C03633=1044.211,253.649,394.364,171.588,39.831,157.569
C03634=1044.205,253.401,394.394,171.585,39.829,157.568
C03635=1044.198,253.153,394.423,171.583,39.827,157.567
C03636=1044.192,252.904,394.453,171.579,39.824,157.567
C03637=1044.185,252.656,394.482,171.576,39.822,157.566
C03638=1044.179,252.408,394.511,171.574,39.820,157.566
C03639=1044.171,252.160,394.540,171.571,39.817,157.565
C03640=1044.165,251.912,394.569,171.568,39.815,157.564
C03641=1044.159,251.664,394.598,171.566,39.812,157.564
C03642=1044.152,251.416,394.627,171.563,39.810,157.563
C03643=1044.146,251.167,394.657,171.561,39.808,157.563
C03644=1044.139,250.919,394.686,171.557,39.806,157.562
C03645=1044.133,250.671,394.715,171.554,39.803,157.561
C03646=1044.126,250.422,394.744,171.552,39.801,157.561
C03647=1044.120,250.174,394.773,171.549,39.798,157.560
C03648=1044.113,249.926,394.802,171.546,39.796,157.560
C03649=1044.107,249.678,394.831,171.544,39.794,157.559
C03650=1044.100,249.430,394.860,171.541,39.791,157.558
C03651=1044.093,249.147,394.894,171.539,39.789,157.558
C03652=1044.085,248.864,394.926,171.535,39.786,157.557
C03653=1044.078,248.581,394.960,171.532,39.784,157.556
C03654=1044.071,248.298,394.992,171.530,39.781,157.556
C03655=1044.064,248.050,395.022,171.527,39.778,157.555
C03656=1044.058,247.802,395.051,171.523,39.776,157.554
C03657=1044.052,247.554,395.080,171.521,39.773,157.554
C03658=1044.046,247.305,395.109,171.518,39.771,157.553
C03659=1044.039,247.057,395.138,171.515,39.769,157.553
C03660=1044.032,246.809,395.166,171.513,39.767,157.552
C03661=1044.025,246.561,395.196,171.510,39.764,157.551
C03662=1044.019,246.313,395.225,171.508,39.762,157.551
C03663=1044.013,246.064,395.254,171.505,39.759,157.550
C03664=1044.007,245.816,395.282,171.502,39.757,157.550
C03665=1044.001,245.568,395.311,171.500,39.755,157.549
C03666=1043.994,245.320,395.339,171.497,39.752,157.548
C03667=1043.987,245.071,395.369,171.495,39.750,157.548
C03668=1043.981,244.823,395.398,171.492,39.747,157.547
C03669=1043.974,244.574,395.426,171.489,39.745,157.547
C03670=1043.968,244.326,395.455,171.487,39.743,157.546
C03671=1043.961,244.078,395.484,171.484,39.741,157.545
C03672=1043.955,243.830,395.511,171.482,39.738,157.545
C03673=1043.949,243.581,395.540,171.479,39.736,157.544
C03674=1043.941,243.333,395.569,171.477,39.734,157.544
C03675=1043.935,243.085,395.598,171.474,39.731,157.543
C03676=1043.929,242.836,395.627,171.471,39.729,157.542
C03677=1043.922,242.588,395.655,171.469,39.726,157.542
C03678=1043.916,242.340,395.683,171.466,39.724,157.541
C03679=1043.909,242.092,395.712,171.464,39.722,157.541
C03680=1043.903,241.844,395.741,171.461,39.720,157.540
C03681=1043.896,241.595,395.769,171.458,39.717,157.539
C03682=1043.890,241.347,395.798,171.456,39.715,157.539
C03683=1043.883,241.099,395.827,171.453,39.713,157.538
C03684=1043.876,240.850,395.855,171.451,39.711,157.538
C03685=1043.869,240.602,395.883,171.448,39.708,157.537
C03686=1043.863,240.353,395.912,171.445,39.706,157.537
C03687=1043.856,240.105,395.940,171.443,39.704,157.536
C03688=1043.850,239.857,395.968,171.440,39.701,157.535
C03689=1043.844,239.608,395.996,171.438,39.699,157.535
C03690=1043.837,239.360,396.024,171.435,39.696,157.534
C03691=1043.830,239.112,396.052,171.432,39.694,157.534
C03692=1043.824,238.864,396.081,171.430,39.692,157.533
C03693=1043.817,238.615,396.109,171.427,39.690,157.532
C03694=1043.810,238.367,396.137,171.425,39.687,157.532
C03695=1043.804,238.119,396.166,171.422,39.685,157.531
C03696=1043.797,237.870,396.194,171.420,39.683,157.531
C03697=1043.790,237.622,396.222,171.417,39.680,157.530
C03698=1043.784,237.373,396.251,171.415,39.678,157.530
C03699=1043.777,237.125,396.279,171.413,39.676,157.529
C03700=1043.770,236.877,396.307,171.410,39.674,157.528
C03701=1043.764,236.628,396.335,171.408,39.671,157.528
C03702=1043.757,236.380,396.364,171.405,39.669,157.527
C03703=1043.751,236.132,396.391,171.403,39.667,157.527
C03704=1043.744,235.883,396.419,171.400,39.665,157.526
C03705=1043.738,235.635,396.447,171.397,39.662,157.526
C03706=1043.731,235.387,396.476,171.395,39.660,157.525
C03707=1043.724,235.098,396.508,171.392,39.657,157.524
C03708=1043.716,234.809,396.541,171.390,39.655,157.524
C03709=1043.708,234.520,396.573,171.386,39.652,157.523
C03710=1043.701,234.232,396.606,171.383,39.649,157.522
C03711=1043.695,233.984,396.634,171.381,39.647,157.522
C03712=1043.688,233.736,396.661,171.378,39.645,157.521
C03713=1043.681,233.488,396.690,171.377,39.642,157.521
C03714=1043.675,233.239,396.718,171.374,39.640,157.520
C03715=1043.668,232.991,396.746,171.371,39.638,157.519
C03716=1043.662,232.742,396.774,171.369,39.635,157.519
C03717=1043.655,232.494,396.801,171.366,39.633,157.518
C03718=1043.649,232.245,396.830,171.364,39.631,157.518
C03719=1043.642,231.997,396.858,171.361,39.629,157.517
C03720=1043.635,231.749,396.886,171.359,39.626,157.517
C03721=1043.629,231.500,396.914,171.357,39.624,157.516
C03722=1043.622,231.252,396.941,171.354,39.622,157.515
C03723=1043.615,231.003,396.969,171.352,39.619,157.515
C03724=1043.609,230.756,396.996,171.349,39.617,157.514
C03725=1043.603,230.507,397.024,171.347,39.615,157.514
C03726=1043.597,230.258,397.053,171.344,39.613,157.513
C03727=1043.590,230.010,397.080,171.342,39.610,157.513
C03728=1043.583,229.762,397.108,171.340,39.608,157.512
C03729=1043.577,229.513,397.136,171.337,39.606,157.512
C03730=1043.570,229.265,397.163,171.335,39.603,157.511
C03731=1043.563,229.016,397.191,171.332,39.601,157.510
C03732=1043.557,228.768,397.219,171.330,39.599,157.510
C03733=1043.550,228.520,397.246,171.327,39.597,157.509
C03734=1043.544,228.272,397.274,171.325,39.594,157.509
C03735=1043.537,228.023,397.302,171.323,39.592,157.508
C03736=1043.530,227.775,397.329,171.321,39.590,157.508
C03737=1043.524,227.526,397.356,171.318,39.587,157.507
C03738=1043.517,227.277,397.384,171.315,39.585,157.506
C03739=1043.511,227.029,397.412,171.313,39.583,157.506
C03740=1043.503,226.781,397.439,171.310,39.581,157.505
C03741=1043.497,226.533,397.466,171.309,39.578,157.505
C03742=1043.491,226.284,397.494,171.306,39.576,157.504
C03743=1043.484,226.035,397.521,171.304,39.574,157.504
C03744=1043.477,225.787,397.549,171.301,39.571,157.503
C03745=1043.471,225.539,397.577,171.298,39.569,157.502
C03746=1043.464,225.290,397.604,171.297,39.567,157.502
C03747=1043.457,225.042,397.632,171.294,39.564,157.501
C03748=1043.451,224.794,397.658,171.292,39.562,157.501
C03749=1043.444,224.545,397.686,171.289,39.560,157.500
C03750=1043.438,224.297,397.714,171.287,39.558,157.500
C03751=1043.431,224.048,397.741,171.285,39.555,157.499
C03752=1043.424,223.799,397.768,171.283,39.553,157.498
C03753=1043.418,223.551,397.796,171.280,39.551,157.498
C03754=1043.412,223.303,397.823,171.277,39.548,157.497
C03755=1043.405,223.054,397.850,171.275,39.546,157.497
C03756=1043.398,222.806,397.878,171.273,39.544,157.496
C03757=1043.392,222.558,397.905,171.271,39.541,157.496
C03758=1043.385,222.309,397.932,171.268,39.539,157.495
C03759=1043.379,222.061,397.960,171.266,39.537,157.495
C03760=1043.372,221.812,397.987,171.264,39.534,157.494
C03761=1043.366,221.564,398.014,171.262,39.532,157.493
C03762=1043.360,221.315,398.042,171.259,39.530,157.493
C03763=1043.352,221.020,398.074,171.256,39.527,157.492
C03764=1043.344,220.723,398.107,171.254,39.524,157.491
C03765=1043.336,220.427,398.139,171.251,39.522,157.491
C03766=1043.329,220.131,398.171,171.248,39.519,157.490
C03767=1043.321,219.883,398.198,171.246,39.517,157.490
C03768=1043.315,219.634,398.225,171.243,39.514,157.489
C03769=1043.308,219.386,398.252,171.242,39.512,157.488
C03770=1043.302,219.137,398.279,171.239,39.510,157.488
C03771=1043.295,218.889,398.307,171.237,39.507,157.487
C03772=1043.288,218.640,398.333,171.234,39.505,157.487
C03773=1043.282,218.392,398.361,171.233,39.503,157.486
C03774=1043.275,218.144,398.387,171.230,39.500,157.486
C03775=1043.268,217.895,398.414,171.227,39.498,157.485
C03776=1043.262,217.646,398.442,171.226,39.496,157.485
C03777=1043.255,217.398,398.468,171.223,39.493,157.484
C03778=1043.248,217.150,398.496,171.221,39.492,157.484
C03779=1043.241,216.901,398.522,171.218,39.489,157.483
C03780=1043.235,216.653,398.549,171.217,39.487,157.482
C03781=1043.229,216.404,398.576,171.214,39.485,157.482
C03782=1043.222,216.155,398.603,171.212,39.483,157.481
C03783=1043.216,215.907,398.630,171.210,39.480,157.481
C03784=1043.209,215.659,398.657,171.208,39.478,157.480
C03785=1043.202,215.410,398.684,171.205,39.476,157.480
C03786=1043.196,215.162,398.710,171.203,39.473,157.479
C03787=1043.189,214.913,398.737,171.201,39.471,157.479
C03788=1043.182,214.665,398.764,171.198,39.469,157.478
C03789=1043.176,214.416,398.791,171.197,39.466,157.477
C03790=1043.169,214.168,398.818,171.194,39.464,157.477
C03791=1043.163,213.920,398.844,171.192,39.462,157.476
C03792=1043.156,213.671,398.871,171.190,39.459,157.476
C03793=1043.149,213.422,398.898,171.188,39.457,157.475
C03794=1043.143,213.174,398.925,171.185,39.455,157.475
C03795=1043.136,212.925,398.952,171.184,39.452,157.474
C03796=1043.130,212.677,398.978,171.181,39.450,157.473
C03797=1043.123,212.428,399.005,171.178,39.448,157.473
C03798=1043.117,212.180,399.032,171.177,39.445,157.472
C03799=1043.111,211.932,399.059,171.174,39.442,157.472
C03800=1043.104,211.683,399.085,171.172,39.440,157.471
C03801=1043.097,211.435,399.111,171.170,39.438,157.471
C03802=1043.091,211.186,399.138,171.168,39.435,157.470
C03803=1043.084,210.938,399.165,171.166,39.433,157.469
C03804=1043.078,210.689,399.192,171.163,39.431,157.469
C03805=1043.071,210.440,399.219,171.161,39.429,157.468
C03806=1043.064,210.192,399.245,171.160,39.427,157.468
C03807=1043.058,209.943,399.272,171.157,39.424,157.467
C03808=1043.051,209.695,399.298,171.154,39.422,157.467
C03809=1043.045,209.446,399.325,171.153,39.420,157.466
C03810=1043.038,209.198,399.351,171.150,39.417,157.466
C03811=1043.031,208.949,399.377,171.149,39.415,157.465
C03812=1043.024,208.701,399.404,171.146,39.413,157.465
C03813=1043.018,208.452,399.430,171.144,39.410,157.464
C03814=1043.011,208.204,399.457,171.142,39.408,157.463
C03815=1043.005,207.955,399.483,171.140,39.406,157.463
C03816=1042.998,207.706,399.510,171.138,39.403,157.462
C03817=1042.992,207.458,399.536,171.136,39.401,157.462
C03818=1042.985,207.210,399.562,171.133,39.399,157.461
C03819=1042.978,206.919,399.593,171.130,39.396,157.461
C03820=1042.970,206.629,399.624,171.129,39.393,157.460
C03821=1042.962,206.338,399.654,171.126,39.391,157.459
C03822=1042.953,206.047,399.685,171.123,39.388,157.459
C03823=1042.927,204.996,399.792,170.852,39.286,157.429
C03824=1042.921,204.748,399.817,170.849,39.284,157.428
C03825=1042.915,204.499,399.843,170.846,39.282,157.428
C03826=1042.909,204.250,399.867,170.843,39.281,157.428
C03827=1042.903,204.002,399.892,170.840,39.279,157.427
C03828=1042.897,203.753,399.918,170.837,39.278,157.427
C03829=1042.891,203.504,399.943,170.835,39.276,157.426
C03830=1042.885,203.256,399.968,170.831,39.275,157.426
C03831=1042.879,203.006,399.993,170.829,39.273,157.426
C03832=1042.873,202.758,400.018,170.826,39.271,157.425
C03833=1042.867,202.510,400.043,170.823,39.270,157.425
C03834=1042.861,202.261,400.068,170.820,39.269,157.424
C03835=1042.854,202.012,400.092,170.817,39.267,157.424
C03836=1042.848,201.763,400.118,170.814,39.265,157.423
C03837=1042.842,201.515,400.143,170.812,39.264,157.423
C03838=1042.835,201.266,400.168,170.808,39.263,157.423
C03839=1042.830,201.017,400.193,170.806,39.261,157.422
C03840=1042.824,200.769,400.218,170.803,39.259,157.422
C03841=1042.817,200.520,400.242,170.800,39.258,157.422
C03842=1042.811,200.271,400.267,170.797,39.256,157.421
C03843=1042.804,200.023,400.292,170.794,39.255,157.421
C03844=1042.798,199.773,400.317,170.791,39.254,157.420
C03845=1042.792,199.526,400.341,170.789,39.252,157.420
C03846=1042.786,199.277,400.366,170.787,39.251,157.420
C03847=1042.780,199.028,400.391,170.783,39.249,157.419
C03848=1042.773,198.779,400.415,170.781,39.248,157.419
C03849=1042.767,198.530,400.441,170.777,39.247,157.419
C03850=1042.761,198.282,400.464,170.775,39.245,157.418
C03851=1042.755,198.033,400.490,170.772,39.244,157.418
C03852=1042.749,197.784,400.514,170.769,39.242,157.417
C03853=1042.742,197.536,400.539,170.766,39.241,157.417
C03854=1042.736,197.286,400.564,170.764,39.239,157.417
C03855=1042.730,197.039,400.588,170.760,39.238,157.416
C03856=1042.724,196.789,400.613,170.758,39.237,157.416
C03857=1042.717,196.541,400.637,170.755,39.235,157.415
C03858=1042.711,196.292,400.662,170.752,39.234,157.415
C03859=1042.706,196.043,400.686,170.749,39.232,157.415
C03860=1042.699,195.795,400.711,170.747,39.231,157.414
C03861=1042.693,195.545,400.735,170.744,39.229,157.414
C03862=1042.687,195.297,400.759,170.741,39.228,157.414
C03863=1042.681,195.049,400.784,170.739,39.227,157.413
C03864=1042.674,194.800,400.809,170.735,39.225,157.413
C03865=1042.668,194.551,400.834,170.733,39.224,157.413
C03866=1042.662,194.303,400.858,170.730,39.222,157.412
C03867=1042.656,194.053,400.882,170.727,39.221,157.412
C03868=1042.650,193.805,400.907,170.725,39.220,157.411
C03869=1042.644,193.556,400.931,170.722,39.219,157.411
C03870=1042.638,193.307,400.956,170.719,39.217,157.411
C03871=1042.631,193.058,400.980,170.716,39.216,157.410
C03872=1042.625,192.810,401.005,170.714,39.214,157.410
C03873=1042.619,192.561,401.029,170.711,39.213,157.410
C03874=1042.613,192.313,401.053,170.708,39.211,157.409
C03875=1042.607,192.064,401.077,170.706,39.210,157.409
C03876=1042.601,191.815,401.102,170.702,39.209,157.409
C03877=1042.595,191.567,401.126,170.700,39.207,157.408
C03878=1042.589,191.317,401.151,170.697,39.206,157.408
C03879=1042.582,191.068,401.175,170.694,39.205,157.407
C03880=1042.577,190.820,401.199,170.692,39.203,157.407
C03881=1042.570,190.571,401.224,170.689,39.202,157.407
C03882=1042.564,190.323,401.248,170.686,39.200,157.406
C03883=1042.558,190.074,401.272,170.684,39.199,157.406
C03884=1042.552,189.789,401.300,170.680,39.198,157.406
C03885=1042.545,189.505,401.328,170.677,39.196,157.405
C03886=1042.538,189.220,401.355,170.675,39.194,157.405
C03887=1042.530,188.936,401.383,170.671,39.193,157.404
C03888=1042.525,188.688,401.407,170.669,39.191,157.404
C03889=1042.518,188.439,401.431,170.666,39.190,157.404
C03890=1042.513,188.190,401.456,170.663,39.189,157.403
C03891=1042.506,187.941,401.480,170.661,39.188,157.403
C03892=1042.501,187.692,401.504,170.658,39.186,157.403
C03893=1042.495,187.443,401.528,170.655,39.185,157.402
C03894=1042.489,187.195,401.552,170.653,39.183,157.402
C03895=1042.483,186.946,401.576,170.650,39.182,157.402
C03896=1042.477,186.697,401.600,170.647,39.181,157.401
C03897=1042.471,186.448,401.625,170.645,39.179,157.401
C03898=1042.465,186.200,401.649,170.642,39.178,157.401
C03899=1042.459,185.951,401.673,170.639,39.177,157.400
C03900=1042.453,185.702,401.697,170.637,39.175,157.400
C03901=1042.447,185.453,401.721,170.634,39.174,157.399
C03902=1042.442,185.205,401.745,170.631,39.173,157.399
C03903=1042.435,184.956,401.769,170.629,39.172,157.399
C03904=1042.429,184.707,401.793,170.626,39.170,157.398
C03905=1042.423,184.458,401.818,170.624,39.169,157.398
C03906=1042.417,184.210,401.841,170.621,39.167,157.398
C03907=1042.412,183.961,401.866,170.619,39.166,157.397
C03908=1042.405,183.712,401.890,170.616,39.165,157.397
C03909=1042.399,183.463,401.913,170.613,39.163,157.397
C03910=1042.393,183.214,401.937,170.611,39.162,157.396
C03911=1042.387,182.966,401.960,170.608,39.161,157.396
C03912=1042.380,182.717,401.984,170.605,39.160,157.396
C03913=1042.374,182.468,402.007,170.603,39.159,157.395
C03914=1042.368,182.219,402.031,170.600,39.158,157.395
C03915=1042.362,181.971,402.055,170.598,39.157,157.395
C03916=1042.355,181.721,402.078,170.595,39.156,157.395
C03917=1042.349,181.473,402.102,170.592,39.154,157.394
C03918=1042.342,181.224,402.126,170.590,39.153,157.394
C03919=1042.337,180.975,402.149,170.587,39.152,157.394
C03920=1042.330,180.726,402.173,170.584,39.151,157.393
C03921=1042.324,180.478,402.197,170.582,39.150,157.393
C03922=1042.318,180.228,402.220,170.580,39.149,157.393
C03923=1042.311,179.980,402.243,170.576,39.148,157.392
C03924=1042.305,179.731,402.266,170.574,39.146,157.392
C03925=1042.299,179.482,402.290,170.572,39.145,157.392
C03926=1042.292,179.233,402.314,170.569,39.144,157.392
C03927=1042.286,178.985,402.337,170.566,39.143,157.391
C03928=1042.280,178.736,402.361,170.564,39.141,157.391
C03929=1042.274,178.487,402.384,170.561,39.140,157.391
C03930=1042.268,178.238,402.407,170.558,39.139,157.390
C03931=1042.262,177.989,402.431,170.556,39.138,157.390
C03932=1042.255,177.741,402.454,170.554,39.137,157.390
C03933=1042.248,177.491,402.477,170.551,39.136,157.389
C03934=1042.242,177.243,402.501,170.548,39.135,157.389
C03935=1042.237,176.994,402.524,170.546,39.134,157.389
C03936=1042.230,176.745,402.548,170.543,39.133,157.388
C03937=1042.224,176.496,402.571,170.540,39.132,157.388
C03938=1042.218,176.248,402.594,170.538,39.131,157.388
C03939=1042.212,175.998,402.618,170.536,39.129,157.388
C03940=1042.206,175.750,402.641,170.533,39.128,157.387
C03941=1042.200,175.500,402.665,170.530,39.127,157.387
C03942=1042.193,175.253,402.688,170.528,39.126,157.387
C03943=1042.187,175.004,402.711,170.526,39.125,157.386
C03944=1042.181,174.754,402.734,170.522,39.123,157.386
C03945=1042.175,174.506,402.758,170.520,39.122,157.386
C03946=1042.169,174.257,402.781,170.518,39.121,157.385
C03947=1042.163,174.009,402.804,170.516,39.120,157.385
C03948=1042.155,173.723,402.830,170.512,39.119,157.385
C03949=1042.149,173.438,402.857,170.510,39.118,157.385
C03950=1042.142,173.153,402.884,170.507,39.116,157.384
C03951=1042.135,172.869,402.910,170.503,39.115,157.384
C03952=1042.129,172.620,402.934,170.501,39.114,157.383
C03953=1042.122,172.371,402.957,170.499,39.113,157.383
C03954=1042.117,172.122,402.980,170.497,39.112,157.383
C03955=1042.110,171.874,403.003,170.494,39.111,157.383
C03956=1042.104,171.625,403.026,170.491,39.110,157.382
C03957=1042.098,171.375,403.049,170.489,39.109,157.382
C03958=1042.092,171.126,403.072,170.487,39.108,157.382
C03959=1042.086,170.878,403.096,170.484,39.107,157.381
C03960=1042.080,170.629,403.119,170.481,39.105,157.381
C03961=1042.074,170.380,403.142,170.479,39.104,157.381
C03962=1042.067,170.131,403.164,170.477,39.103,157.381
C03963=1042.061,169.883,403.188,170.474,39.102,157.380
C03964=1042.056,169.634,403.211,170.472,39.100,157.380
C03965=1042.049,169.384,403.234,170.470,39.099,157.380
C03966=1042.044,169.135,403.257,170.466,39.098,157.379
C03967=1042.038,168.887,403.280,170.464,39.097,157.379
C03968=1042.031,168.639,403.303,170.462,39.096,157.379
C03969=1042.025,168.390,403.326,170.460,39.095,157.378
C03970=1042.020,168.141,403.349,170.457,39.094,157.378
C03971=1042.013,167.891,403.373,170.454,39.093,157.378
C03972=1042.008,167.642,403.396,170.452,39.092,157.378
C03973=1042.002,167.393,403.418,170.449,39.091,157.377
C03974=1041.995,167.145,403.441,170.447,39.089,157.377
C03975=1041.989,166.897,403.464,170.445,39.088,157.377
C03976=1041.984,166.648,403.487,170.443,39.087,157.376
C03977=1041.978,166.399,403.510,170.439,39.086,157.376
C03978=1041.972,166.149,403.534,170.437,39.085,157.376
C03979=1041.965,165.901,403.556,170.435,39.084,157.376
C03980=1041.959,165.652,403.579,170.433,39.083,157.375
C03981=1041.954,165.403,403.602,170.430,39.082,157.375
C03982=1041.948,165.154,403.625,170.428,39.081,157.375
C03983=1041.942,164.905,403.648,170.426,39.079,157.374
C03984=1041.936,164.656,403.670,170.423,39.078,157.374
C03985=1041.930,164.408,403.693,170.420,39.077,157.374
C03986=1041.924,164.159,403.716,170.418,39.076,157.373
C03987=1041.919,163.910,403.739,170.416,39.075,157.373
C03988=1041.913,163.661,403.762,170.414,39.074,157.373
C03989=1041.906,163.412,403.785,170.411,39.073,157.373
C03990=1041.900,163.163,403.808,170.409,39.072,157.372
C03991=1041.894,162.914,403.831,170.407,39.071,157.372
C03992=1041.889,162.665,403.853,170.403,39.070,157.372
C03993=1041.883,162.416,403.876,170.401,39.068,157.371
C03994=1041.876,162.167,403.899,170.399,39.067,157.371
C03995=1041.871,161.918,403.922,170.397,39.066,157.371
C03996=1041.865,161.670,403.945,170.394,39.065,157.371
C03997=1041.859,161.421,403.968,170.392,39.064,157.370
C03998=1041.853,161.172,403.990,170.390,39.063,157.370
C03999=1041.847,160.923,404.012,170.388,39.062,157.370
C04000=1041.842,160.674,404.035,170.385,39.061,157.369
C04001=1041.836,160.425,404.058,170.383,39.060,157.369
C04002=1041.829,160.176,404.080,170.380,39.059,157.369
C04003=1041.824,159.927,404.103,170.378,39.058,157.369
C04004=1041.817,159.678,404.125,170.375,39.057,157.368
C04005=1041.812,159.429,404.148,170.373,39.056,157.368
C04006=1041.805,159.181,404.170,170.371,39.055,157.368
C04007=1041.799,158.932,404.193,170.369,39.054,157.368
C04008=1041.793,158.683,404.215,170.367,39.053,157.367
C04009=1041.787,158.434,404.237,170.364,39.052,157.367
C04010=1041.781,158.185,404.260,170.361,39.051,157.367
C04011=1041.775,157.936,404.282,170.359,39.050,157.367
C04012=1041.766,157.610,404.311,170.357,39.049,157.366
C04013=1041.758,157.283,404.341,170.353,39.048,157.366
C04014=1041.751,156.956,404.370,170.350,39.046,157.366
C04015=1041.742,156.630,404.399,170.347,39.045,157.365
C04016=1041.737,156.381,404.422,170.344,39.044,157.365
C04017=1041.730,156.132,404.444,170.342,39.043,157.365
C04018=1041.724,155.884,404.466,170.340,39.042,157.364
C04019=1041.718,155.634,404.489,170.338,39.041,157.364
C04020=1041.712,155.385,404.511,170.335,39.040,157.364
C04021=1041.706,155.136,404.533,170.333,39.039,157.364
C04022=1041.700,154.887,404.556,170.331,39.038,157.363
C04023=1041.694,154.639,404.578,170.328,39.037,157.363
C04024=1041.687,154.390,404.600,170.325,39.036,157.363
C04025=1041.682,154.141,404.623,170.323,39.035,157.363
C04026=1041.676,153.891,404.644,170.321,39.035,157.362
C04027=1041.669,153.643,404.666,170.319,39.033,157.362
C04028=1041.663,153.394,404.688,170.317,39.032,157.362
C04029=1041.657,153.145,404.711,170.314,39.032,157.362
C04030=1041.651,152.896,404.733,170.312,39.031,157.361
C04031=1041.645,152.647,404.755,170.310,39.030,157.361
C04032=1041.638,152.398,404.777,170.308,39.028,157.361
C04033=1041.632,152.149,404.799,170.306,39.028,157.361
C04034=1041.627,151.900,404.821,170.303,39.027,157.360
C04035=1041.621,151.651,404.843,170.300,39.026,157.360
C04036=1041.614,151.403,404.865,170.298,39.025,157.360
C04037=1041.608,151.153,404.887,170.296,39.024,157.360
C04038=1041.602,150.905,404.909,170.293,39.023,157.359
C04039=1041.596,150.655,404.931,170.291,39.023,157.359
C04040=1041.590,150.407,404.953,170.289,39.021,157.359
C04041=1041.584,150.157,404.975,170.287,39.020,157.359
C04042=1041.578,149.908,404.997,170.284,39.019,157.358
C04043=1041.571,149.660,405.019,170.282,39.019,157.358
C04044=1041.566,149.410,405.041,170.280,39.018,157.358
C04045=1041.560,149.162,405.063,170.278,39.016,157.358
C04046=1041.554,148.913,405.085,170.276,39.016,157.357
C04047=1041.548,148.664,405.107,170.273,39.015,157.357
C04048=1041.542,148.436,405.127,170.271,39.014,157.357
C04049=1041.536,148.207,405.147,170.269,39.013,157.357
C04050=1041.531,147.978,405.167,170.267,39.013,157.357
C04051=1041.525,147.750,405.187,170.265,39.012,157.356
C04052=1041.519,147.521,405.208,170.262,39.010,157.356
C04053=1041.514,147.293,405.227,170.260,39.010,157.356
C04054=1041.508,147.065,405.247,170.259,39.009,157.356
C04055=1041.503,146.837,405.267,170.257,39.008,157.355
C04056=1041.497,146.588,405.288,170.255,39.007,157.355
C04057=1041.490,146.338,405.310,170.252,39.007,157.355
C04058=1041.484,146.089,405.332,170.250,39.006,157.355
C04059=1041.478,145.841,405.354,170.247,39.005,157.355
C04060=1041.472,145.591,405.376,170.245,39.004,157.354
C04061=1041.466,145.343,405.397,170.243,39.004,157.354
C04062=1041.460,145.094,405.419,170.240,39.002,157.354
C04063=1041.454,144.845,405.440,170.238,39.001,157.354
C04064=1041.448,144.595,405.462,170.236,39.001,157.353
C04065=1041.441,144.347,405.484,170.234,39.000,157.353
C04066=1041.435,144.098,405.506,170.232,38.999,157.353
C04067=1041.429,143.849,405.527,170.229,38.998,157.353
C04068=1041.423,143.600,405.549,170.227,38.997,157.352
C04069=1041.417,143.351,405.570,170.225,38.996,157.352
C04070=1041.410,143.102,405.591,170.223,38.995,157.352
C04071=1041.404,142.853,405.613,170.221,38.995,157.352
C04072=1041.398,142.604,405.634,170.218,38.994,157.351
C04073=1041.392,142.355,405.656,170.216,38.993,157.351
C04074=1041.386,142.106,405.678,170.214,38.992,157.351
C04075=1041.380,141.856,405.699,170.212,38.991,157.351
C04076=1041.373,141.571,405.724,170.209,38.990,157.351
C04077=1041.366,141.286,405.750,170.206,38.989,157.350
C04078=1041.359,141.000,405.773,170.204,38.988,157.350
C04079=1041.352,140.714,405.799,170.202,38.987,157.350
C04080=1041.346,140.465,405.820,170.200,38.987,157.350
C04081=1041.340,140.217,405.841,170.197,38.986,157.349
C04082=1041.334,139.967,405.863,170.195,38.984,157.349
C04083=1041.328,139.718,405.885,170.193,38.984,157.349
C04084=1041.322,139.469,405.906,170.191,38.983,157.349
C04085=1041.315,139.221,405.927,170.189,38.982,157.348
C04086=1041.309,138.972,405.949,170.186,38.981,157.348
C04087=1041.303,138.722,405.970,170.184,38.981,157.348
C04088=1041.297,138.473,405.991,170.182,38.980,157.348
C04089=1041.291,138.224,406.012,170.180,38.979,157.348
C04090=1041.285,137.975,406.034,170.177,38.978,157.347
C04091=1041.279,137.726,406.055,170.175,38.977,157.347
C04092=1041.272,137.477,406.077,170.173,38.976,157.347
C04093=1041.266,137.229,406.097,170.171,38.976,157.347
C04094=1041.260,136.979,406.119,170.169,38.975,157.346
C04095=1041.254,136.730,406.140,170.167,38.974,157.346
C04096=1041.249,136.481,406.161,170.164,38.973,157.346
C04097=1041.242,136.232,406.182,170.162,38.973,157.346
C04098=1041.236,135.983,406.204,170.160,38.971,157.345
C04099=1041.229,135.734,406.226,170.158,38.971,157.345
C04100=1041.223,135.485,406.246,170.156,38.970,157.345
C04101=1041.217,135.236,406.267,170.153,38.969,157.345
C04102=1041.211,134.987,406.289,170.151,38.968,157.345
C04103=1041.205,134.738,406.309,170.149,38.968,157.344
C04104=1041.199,134.489,406.331,170.147,38.966,157.344
C04105=1041.193,134.239,406.352,170.145,38.966,157.344
C04106=1041.186,133.991,406.373,170.142,38.965,157.344
C04107=1041.180,133.742,406.394,170.140,38.964,157.344
C04108=1041.174,133.492,406.415,170.138,38.963,157.343
C04109=1041.168,133.244,406.436,170.136,38.963,157.343
C04110=1041.162,132.995,406.458,170.134,38.962,157.343
C04111=1041.156,132.745,406.479,170.131,38.961,157.343
C04112=1041.150,132.497,406.499,170.129,38.961,157.343
C04113=1041.144,132.247,406.521,170.127,38.959,157.342
C04114=1041.138,131.999,406.542,170.125,38.959,157.342
C04115=1041.131,131.749,406.562,170.123,38.958,157.342
C04116=1041.125,131.500,406.584,170.121,38.957,157.342
C04117=1041.120,131.252,406.605,170.118,38.956,157.341
C04118=1041.113,131.002,406.626,170.116,38.956,157.341
C04119=1041.107,130.753,406.647,170.114,38.955,157.341
C04120=1041.101,130.504,406.667,170.112,38.954,157.341
C04121=1041.094,130.255,406.688,170.110,38.954,157.341
C04122=1041.088,130.005,406.709,170.107,38.952,157.340
C04123=1041.082,129.757,406.730,170.105,38.952,157.340
C04124=1041.075,129.508,406.750,170.103,38.951,157.340
C04125=1041.069,129.259,406.772,170.101,38.950,157.340
C04126=1041.063,129.010,406.792,170.099,38.950,157.340
C04127=1041.056,128.761,406.813,170.097,38.949,157.339
C04128=1041.050,128.511,406.834,170.095,38.948,157.339
C04129=1041.044,128.263,406.854,170.093,38.948,157.339
C04130=1041.038,128.013,406.875,170.091,38.947,157.339
C04131=1041.032,127.765,406.896,170.089,38.946,157.339
C04132=1041.025,127.515,406.916,170.087,38.945,157.338
C04133=1041.018,127.266,406.937,170.085,38.945,157.338
C04134=1041.013,127.017,406.958,170.082,38.944,157.338
C04135=1041.006,126.768,406.979,170.080,38.943,157.338
C04136=1041.000,126.520,406.999,170.078,38.943,157.338
C04137=1040.994,126.270,407.021,170.076,38.942,157.337
C04138=1040.988,126.021,407.041,170.074,38.941,157.337
C04139=1040.982,125.772,407.061,170.071,38.941,157.337
C04140=1040.975,125.486,407.085,170.069,38.940,157.337
C04141=1040.968,125.200,407.109,170.066,38.939,157.337
C04142=1040.961,124.915,407.133,170.064,38.938,157.336
C04143=1040.953,124.628,407.156,170.062,38.938,157.336
C04144=1040.947,124.380,407.177,170.059,38.936,157.336
C04145=1040.940,124.130,407.197,170.057,38.936,157.336
C04146=1040.935,123.881,407.218,170.055,38.935,157.335
C04147=1040.928,123.632,407.239,170.053,38.934,157.335
C04148=1040.922,123.384,407.259,170.051,38.934,157.335
C04149=1040.916,123.134,407.280,170.049,38.933,157.335
C04150=1040.910,122.886,407.300,170.046,38.932,157.335
C04151=1040.904,122.636,407.321,170.044,38.932,157.335
C04152=1040.898,122.387,407.341,170.043,38.930,157.334
C04153=1040.891,122.138,407.362,170.041,38.930,157.334
C04154=1040.885,121.889,407.382,170.039,38.929,157.334
C04155=1040.880,121.639,407.403,170.036,38.928,157.334
C04156=1040.874,121.391,407.423,170.034,38.928,157.334
C04157=1040.867,121.142,407.444,170.032,38.927,157.333
C04158=1040.861,120.893,407.464,170.030,38.926,157.333
C04159=1040.855,120.643,407.485,170.028,38.926,157.333
C04160=1040.849,120.394,407.505,170.026,38.924,157.333
C04161=1040.842,120.145,407.526,170.023,38.924,157.332
C04162=1040.837,119.896,407.546,170.021,38.923,157.332
C04163=1040.830,119.647,407.567,170.019,38.922,157.332
C04164=1040.824,119.398,407.587,170.018,38.922,157.332
C04165=1040.819,119.149,407.608,170.016,38.921,157.332
C04166=1040.812,118.900,407.628,170.014,38.920,157.331
C04167=1040.806,118.651,407.648,170.011,38.920,157.331
C04168=1040.799,118.402,407.669,170.009,38.918,157.331
C04169=1040.794,118.152,407.689,170.007,38.918,157.331
C04170=1040.787,117.903,407.710,170.005,38.917,157.331
C04171=1040.781,117.655,407.730,170.003,38.916,157.330
C04172=1040.776,117.406,407.751,170.000,38.916,157.330
C04173=1040.769,117.156,407.771,169.998,38.915,157.330
C04174=1040.763,116.907,407.791,169.997,38.914,157.330
C04175=1040.757,116.658,407.811,169.995,38.914,157.330
C04176=1040.751,116.409,407.832,169.993,38.912,157.329
C04177=1040.745,116.160,407.852,169.991,38.912,157.329
C04178=1040.739,115.910,407.872,169.988,38.911,157.329
C04179=1040.733,115.661,407.892,169.986,38.910,157.329
C04180=1040.727,115.413,407.913,169.984,38.910,157.329
C04181=1040.721,115.163,407.934,169.982,38.909,157.328
C04182=1040.715,114.915,407.954,169.980,38.908,157.328
C04183=1040.709,114.665,407.975,169.979,38.908,157.328
C04184=1040.703,114.416,407.995,169.976,38.906,157.328
C04185=1040.697,114.167,408.015,169.974,38.906,157.328
C04186=1040.690,113.918,408.035,169.972,38.905,157.327
C04187=1040.685,113.669,408.055,169.970,38.904,157.327
C04188=1040.679,113.420,408.075,169.968,38.904,157.327
C04189=1040.672,113.170,408.096,169.965,38.903,157.327
C04190=1040.666,112.921,408.116,169.963,38.902,157.327
C04191=1040.660,112.673,408.136,169.962,38.902,157.326
C04192=1040.654,112.423,408.156,169.960,38.900,157.326
C04193=1040.648,112.174,408.176,169.958,38.900,157.326
C04194=1040.642,111.925,408.196,169.956,38.899,157.326
C04195=1040.636,111.675,408.215,169.953,38.899,157.326
C04196=1040.630,111.426,408.235,169.951,38.898,157.325
C04197=1040.624,111.178,408.255,169.949,38.897,157.325
C04198=1040.617,110.928,408.276,169.947,38.897,157.325
C04199=1040.611,110.679,408.296,169.945,38.896,157.325
C04200=1040.604,110.430,408.316,169.943,38.895,157.325
C04201=1040.598,110.181,408.336,169.941,38.895,157.325
C04202=1040.592,109.932,408.355,169.939,38.894,157.324
C04203=1040.585,109.682,408.375,169.937,38.894,157.324
C04204=1040.579,109.396,408.398,169.935,38.892,157.324
C04205=1040.571,109.111,408.420,169.932,38.892,157.324
C04206=1040.565,108.825,408.443,169.930,38.892,157.324
C04207=1040.557,108.539,408.465,169.927,38.890,157.323
C04208=1040.551,108.289,408.486,169.925,38.890,157.323
C04209=1040.545,108.041,408.506,169.923,38.889,157.323
C04210=1040.539,107.792,408.526,169.921,38.889,157.323
C04211=1040.532,107.542,408.546,169.919,38.888,157.323
C04212=1040.526,107.293,408.565,169.918,38.887,157.322
C04213=1040.520,107.044,408.585,169.916,38.887,157.322
C04214=1040.513,106.795,408.605,169.913,38.886,157.322
C04215=1040.507,106.545,408.624,169.911,38.886,157.322
C04216=1040.501,106.297,408.644,169.909,38.884,157.322
C04217=1040.495,106.048,408.664,169.907,38.884,157.322
C04218=1040.489,105.798,408.684,169.905,38.883,157.321
C04219=1040.482,105.549,408.703,169.903,38.883,157.321
C04220=1040.476,105.300,408.723,169.901,38.882,157.321
C04221=1040.470,105.051,408.743,169.899,38.881,157.321
C04222=1040.464,104.801,408.763,169.897,38.881,157.321
C04223=1040.458,104.553,408.783,169.895,38.880,157.321
C04224=1040.451,104.304,408.802,169.893,38.880,157.320
C04225=1040.445,104.054,408.822,169.891,38.879,157.320
C04226=1040.439,103.805,408.842,169.888,38.878,157.320
C04227=1040.433,103.556,408.861,169.886,38.878,157.320
C04228=1040.427,103.307,408.881,169.885,38.877,157.320
C04229=1040.421,103.058,408.901,169.883,38.876,157.319
C04230=1040.414,102.808,408.920,169.881,38.875,157.319
C04231=1040.408,102.559,408.940,169.879,38.875,157.319
C04232=1040.403,102.310,408.959,169.877,38.874,157.319
C04233=1040.397,102.061,408.979,169.874,38.873,157.319
C04234=1040.391,101.812,408.999,169.872,38.873,157.318
C04235=1040.384,101.563,409.018,169.871,38.872,157.318
C04236=1040.378,101.314,409.038,169.869,38.872,157.318
C04237=1040.372,101.064,409.057,169.867,38.870,157.318
C04238=1040.366,100.815,409.077,169.865,38.870,157.318
C04239=1040.360,100.566,409.096,169.862,38.869,157.318
C04240=1040.353,100.317,409.116,169.860,38.869,157.317
C04241=1040.347,100.067,409.135,169.858,38.868,157.317
C04242=1040.340,99.819,409.155,169.856,38.867,157.317
C04243=1040.335,99.569,409.174,169.855,38.867,157.317
C04244=1040.329,99.321,409.194,169.853,38.866,157.317
C04245=1040.322,99.071,409.213,169.850,38.866,157.317
C04246=1040.316,98.822,409.233,169.848,38.865,157.316
C04247=1040.309,98.573,409.251,169.846,38.865,157.316
C04248=1040.304,98.323,409.271,169.844,38.864,157.316
C04249=1040.297,98.075,409.290,169.842,38.863,157.316
C04250=1040.291,97.825,409.310,169.840,38.862,157.316
C04251=1040.284,97.576,409.329,169.839,38.862,157.316
C04252=1040.278,97.327,409.348,169.836,38.861,157.315
C04253=1040.272,97.078,409.367,169.834,38.861,157.315
C04254=1040.266,96.829,409.387,169.832,38.860,157.315
C04255=1040.259,96.579,409.406,169.830,38.860,157.315
C04256=1040.253,96.330,409.425,169.828,38.859,157.315
C04257=1040.246,96.081,409.444,169.826,38.858,157.314
C04258=1040.241,95.832,409.464,169.824,38.858,157.314
C04259=1040.235,95.582,409.483,169.822,38.857,157.314
C04260=1040.228,95.334,409.502,169.820,38.857,157.314
C04261=1040.223,95.084,409.522,169.818,38.856,157.314
C04262=1040.216,94.835,409.540,169.816,38.856,157.314
C04263=1040.210,94.586,409.561,169.814,38.854,157.313
C04264=1040.203,94.337,409.579,169.812,38.854,157.313
C04265=1040.197,94.087,409.598,169.809,38.853,157.313
C04266=1040.191,93.839,409.618,169.808,38.853,157.313
C04267=1040.185,93.589,409.637,169.806,38.852,157.313
C04268=1040.178,93.303,409.659,169.804,38.851,157.313
C04269=1040.170,93.017,409.681,169.802,38.851,157.312
C04270=1040.163,92.731,409.703,169.799,38.850,157.312
C04271=1040.156,92.445,409.725,169.796,38.849,157.312
C04272=1040.150,92.196,409.744,169.794,38.849,157.312
C04273=1040.144,91.947,409.763,169.793,38.848,157.312
C04274=1040.138,91.697,409.782,169.791,38.847,157.312
C04275=1040.132,91.448,409.801,169.789,38.847,157.311
C04276=1040.126,91.199,409.821,169.787,38.846,157.311
C04277=1040.119,90.950,409.839,169.785,38.845,157.311
C04278=1040.113,90.701,409.859,169.782,38.845,157.311
C04279=1040.107,90.452,409.877,169.781,38.844,157.311
C04280=1040.101,90.202,409.897,169.779,38.844,157.310
C04281=1040.095,89.953,409.915,169.777,38.843,157.310
C04282=1040.088,89.705,409.935,169.775,38.843,157.310
C04283=1040.083,89.455,409.954,169.773,38.842,157.310
C04284=1040.076,89.205,409.973,169.771,38.842,157.310
C04285=1040.069,88.956,409.991,169.769,38.841,157.310
C04286=1040.063,88.707,410.010,169.766,38.840,157.309
C04287=1040.057,88.458,410.029,169.765,38.839,157.309
C04288=1040.051,88.209,410.048,169.763,38.839,157.309
C04289=1040.044,87.959,410.067,169.761,38.838,157.309
C04290=1040.038,87.710,410.085,169.759,38.838,157.309
C04291=1040.031,87.461,410.104,169.757,38.837,157.309
C04292=1040.026,87.212,410.123,169.754,38.837,157.309
C04293=1040.019,86.963,410.142,169.752,38.836,157.308
C04294=1040.013,86.713,410.160,169.750,38.836,157.308
C04295=1040.006,86.464,410.179,169.749,38.835,157.308
C04296=1040.001,86.215,410.198,169.747,38.835,157.308
C04297=1039.994,85.966,410.217,169.745,38.834,157.308
C04298=1039.988,85.717,410.236,169.743,38.834,157.308
C04299=1039.981,85.468,410.254,169.741,38.833,157.307
C04300=1039.975,85.218,410.273,169.738,38.833,157.307
C04301=1039.969,84.969,410.292,169.736,38.832,157.307
C04302=1039.963,84.720,410.311,169.735,38.832,157.307
C04303=1039.956,84.471,410.329,169.733,38.830,157.307
C04304=1039.950,84.222,410.348,169.731,38.830,157.307
C04305=1039.944,83.973,410.367,169.729,38.829,157.306
C04306=1039.938,83.723,410.386,169.727,38.829,157.306
C04307=1039.931,83.474,410.405,169.724,38.828,157.306
C04308=1039.925,83.224,410.423,169.722,38.828,157.306
C04309=1039.919,82.975,410.441,169.721,38.827,157.306
C04310=1039.912,82.726,410.460,169.719,38.827,157.306
C04311=1039.907,82.477,410.479,169.717,38.826,157.306
C04312=1039.900,82.227,410.498,169.715,38.826,157.305
C04313=1039.894,81.978,410.516,169.713,38.825,157.305
C04314=1039.887,81.729,410.535,169.710,38.824,157.305
C04315=1039.881,81.480,410.554,169.709,38.824,157.305
C04316=1039.876,81.230,410.572,169.707,38.823,157.305
C04317=1039.869,80.981,410.591,169.705,38.822,157.304
C04318=1039.863,80.732,410.610,169.703,38.822,157.304
C04319=1039.857,80.483,410.628,169.701,38.821,157.304
C04320=1039.851,80.234,410.647,169.699,38.821,157.304
C04321=1039.844,79.985,410.665,169.696,38.820,157.304
C04322=1039.839,79.735,410.684,169.695,38.820,157.304
C04323=1039.832,79.486,410.702,169.693,38.819,157.303
C04324=1039.826,79.237,410.721,169.691,38.818,157.303
C04325=1039.819,78.988,410.740,169.689,38.818,157.303
C04326=1039.813,78.739,410.758,169.687,38.817,157.303
C04327=1039.807,78.489,410.776,169.685,38.817,157.303
C04328=1039.801,78.239,410.795,169.683,38.816,157.303
C04329=1039.795,77.991,410.814,169.681,38.816,157.303
C04330=1039.789,77.741,410.832,169.679,38.815,157.302
C04331=1039.783,77.492,410.850,169.677,38.815,157.302
C04332=1039.775,77.206,410.871,169.675,38.814,157.302
C04333=1039.768,76.920,410.893,169.673,38.813,157.302
C04334=1039.761,76.634,410.914,169.671,38.812,157.302
C04335=1039.754,76.347,410.935,169.668,38.812,157.302
C04336=1039.747,76.098,410.953,169.666,38.811,157.301
C04337=1039.741,75.849,410.972,169.664,38.811,157.301
C04338=1039.735,75.600,410.990,169.662,38.810,157.301
C04339=1039.729,75.351,411.008,169.660,38.810,157.301
C04340=1039.722,75.102,411.025,169.658,38.809,157.301
C04341=1039.716,74.853,411.044,169.656,38.809,157.301
C04342=1039.709,74.603,411.063,169.654,38.808,157.300
C04343=1039.703,74.354,411.081,169.652,38.808,157.300
C04344=1039.697,74.105,411.099,169.650,38.807,157.300
C04345=1039.691,73.855,411.117,169.648,38.807,157.300
C04346=1039.685,73.606,411.136,169.646,38.806,157.300
C04347=1039.678,73.357,411.154,169.644,38.806,157.300
C04348=1039.672,73.108,411.172,169.642,38.805,157.300
C04349=1039.666,72.858,411.191,169.640,38.805,157.299
C04350=1039.660,72.609,411.209,169.638,38.804,157.299
C04351=1039.652,72.360,411.227,169.636,38.803,157.299
C04352=1039.647,72.111,411.244,169.634,38.803,157.299
C04353=1039.641,71.862,411.263,169.632,38.802,157.299
C04354=1039.634,71.612,411.281,169.630,38.802,157.299
C04355=1039.628,71.363,411.300,169.628,38.801,157.298
C04356=1039.622,71.113,411.317,169.626,38.801,157.298
C04357=1039.615,70.864,411.336,169.625,38.800,157.298
C04358=1039.610,70.615,411.354,169.622,38.800,157.298
C04359=1039.603,70.366,411.372,169.620,38.799,157.298
C04360=1039.597,70.116,411.390,169.618,38.799,157.298
C04361=1039.590,69.867,411.408,169.616,38.798,157.298
C04362=1039.585,69.618,411.426,169.614,38.798,157.297
C04363=1039.579,69.368,411.444,169.613,38.797,157.297
C04364=1039.572,69.119,411.462,169.611,38.797,157.297
C04365=1039.565,68.870,411.480,169.609,38.796,157.297
C04366=1039.559,68.621,411.498,169.606,38.796,157.297
C04367=1039.553,68.372,411.516,169.604,38.795,157.297
C04368=1039.547,68.122,411.534,169.602,38.794,157.297
C04369=1039.540,67.873,411.552,169.600,38.794,157.296
C04370=1039.534,67.623,411.570,169.598,38.793,157.296
C04371=1039.528,67.374,411.588,169.597,38.793,157.296
C04372=1039.521,67.126,411.606,169.595,38.792,157.296
C04373=1039.515,66.876,411.623,169.593,38.792,157.296
C04374=1039.509,66.626,411.641,169.590,38.791,157.296
C04375=1039.503,66.377,411.660,169.588,38.791,157.295
C04376=1039.496,66.128,411.677,169.586,38.790,157.295
C04377=1039.490,65.879,411.695,169.584,38.790,157.295
C04378=1039.484,65.629,411.714,169.583,38.789,157.295
C04379=1039.477,65.380,411.731,169.581,38.789,157.295
C04380=1039.471,65.131,411.749,169.579,38.788,157.295
C04381=1039.465,64.882,411.767,169.576,38.788,157.295
C04382=1039.458,64.632,411.785,169.574,38.787,157.294
C04383=1039.453,64.383,411.802,169.572,38.787,157.294
C04384=1039.447,64.134,411.820,169.570,38.786,157.294
C04385=1039.440,63.884,411.837,169.568,38.786,157.294
C04386=1039.433,63.635,411.856,169.567,38.785,157.294
C04387=1039.426,63.386,411.873,169.565,38.785,157.294
C04388=1039.421,63.137,411.891,169.563,38.785,157.294
C04389=1039.414,62.887,411.908,169.561,38.784,157.293
C04390=1039.407,62.638,411.926,169.558,38.784,157.293
C04391=1039.401,62.388,411.944,169.556,38.783,157.293
C04392=1039.394,62.140,411.961,169.554,38.782,157.293
C04393=1039.388,61.890,411.979,169.552,38.783,157.293
C04394=1039.381,61.641,411.996,169.550,38.782,157.293
C04395=1039.376,61.392,412.014,169.548,38.782,157.293
C04396=1039.368,61.105,412.034,169.546,38.781,157.293
C04397=1039.360,60.819,412.054,169.544,38.781,157.292
C04398=1039.353,60.533,412.074,169.542,38.780,157.292
C04399=1039.346,60.246,412.094,169.539,38.779,157.292
C04400=1039.340,59.997,412.112,169.537,38.779,157.292
C04401=1039.333,59.748,412.129,169.535,38.778,157.292
C04402=1039.326,59.498,412.147,169.533,38.779,157.292
C04403=1039.321,59.249,412.164,169.531,38.778,157.292
C04404=1039.314,59.000,412.181,169.529,38.778,157.291
C04405=1039.307,58.750,412.199,169.527,38.777,157.291
C04406=1039.302,58.501,412.216,169.525,38.776,157.291
C04407=1039.295,58.252,412.234,169.523,38.776,157.291
C04408=1039.289,58.002,412.252,169.521,38.775,157.291
C04409=1039.282,57.753,412.269,169.519,38.776,157.291
C04410=1039.275,57.504,412.286,169.517,38.775,157.291
C04411=1039.269,57.254,412.304,169.515,38.774,157.291
C04412=1039.263,57.005,412.321,169.513,38.774,157.290
C04413=1039.256,56.756,412.338,169.511,38.773,157.290
C04414=1039.250,56.506,412.356,169.509,38.773,157.290
C04415=1039.244,56.258,412.373,169.507,38.772,157.290
C04416=1039.238,56.008,412.391,169.505,38.772,157.290
C04417=1039.231,55.758,412.408,169.503,38.772,157.290
C04418=1039.225,55.510,412.425,169.501,38.771,157.290
C04419=1039.219,55.260,412.443,169.499,38.771,157.289
C04420=1039.212,55.011,412.460,169.497,38.770,157.289
C04421=1039.205,54.762,412.478,169.495,38.770,157.289
C04422=1039.199,54.512,412.496,169.493,38.769,157.289
C04423=1039.193,54.263,412.513,169.491,38.769,157.289
C04424=1039.186,54.014,412.530,169.489,38.768,157.289
C04425=1039.181,53.764,412.547,169.487,38.768,157.289
C04426=1039.174,53.515,412.564,169.485,38.768,157.289
C04427=1039.168,53.265,412.582,169.483,38.767,157.288
C04428=1039.162,53.016,412.599,169.481,38.767,157.288
C04429=1039.155,52.767,412.616,169.479,38.766,157.288
C04430=1039.149,52.518,412.634,169.477,38.766,157.288
C04431=1039.142,52.268,412.651,169.475,38.765,157.288
C04432=1039.137,52.019,412.667,169.473,38.765,157.288
C04433=1039.130,51.769,412.685,169.470,38.764,157.287
C04434=1039.124,51.521,412.702,169.469,38.764,157.287
C04435=1039.117,51.271,412.720,169.467,38.763,157.287
C04436=1039.111,51.021,412.738,169.465,38.763,157.287
C04437=1039.105,50.773,412.755,169.463,38.763,157.287
C04438=1039.098,50.523,412.771,169.461,38.762,157.287
C04439=1039.093,50.274,412.789,169.459,38.762,157.287
C04440=1039.086,50.024,412.806,169.457,38.761,157.287
C04441=1039.080,49.775,412.823,169.455,38.761,157.286
C04442=1039.074,49.525,412.840,169.452,38.760,157.286
C04443=1039.068,49.276,412.857,169.451,38.759,157.286
C04444=1039.061,49.027,412.875,169.449,38.759,157.286
C04445=1039.055,48.778,412.892,169.447,38.758,157.286
C04446=1039.049,48.528,412.909,169.445,38.758,157.286
C04447=1039.042,48.279,412.926,169.443,38.757,157.285
C04448=1039.036,48.029,412.944,169.441,38.757,157.285
C04449=1039.030,47.781,412.961,169.439,38.756,157.285
C04450=1039.024,47.531,412.977,169.436,38.756,157.285
C04451=1039.017,47.282,412.994,169.434,38.755,157.285
C04452=1039.012,47.033,413.012,169.433,38.755,157.285
C04453=1039.005,46.783,413.028,169.431,38.755,157.285
C04454=1038.999,46.534,413.045,169.429,38.754,157.285
C04455=1038.993,46.284,413.063,169.427,38.754,157.284
C04456=1038.987,46.035,413.080,169.425,38.753,157.284
C04457=1038.980,45.786,413.097,169.423,38.753,157.284
C04458=1038.974,45.536,413.115,169.421,38.752,157.284
C04459=1038.969,45.287,413.131,169.418,38.752,157.284
C04460=1038.961,45.001,413.151,169.416,38.751,157.284
C04461=1038.954,44.714,413.170,169.414,38.751,157.284
C04462=1038.947,44.427,413.190,169.412,38.750,157.283
C04463=1038.939,44.141,413.209,169.410,38.749,157.283
C04464=1038.934,43.891,413.226,169.408,38.748,157.283
C04465=1038.927,43.642,413.244,169.406,38.748,157.283
C04466=1038.921,43.393,413.260,169.403,38.747,157.283
C04467=1038.915,43.143,413.278,169.401,38.747,157.283
C04468=1038.909,42.894,413.295,169.399,38.747,157.282
C04469=1038.903,42.645,413.311,169.397,38.746,157.282
C04470=1038.896,42.395,413.328,169.395,38.746,157.282
C04471=1038.890,42.146,413.345,169.394,38.745,157.282
C04472=1038.883,41.897,413.362,169.392,38.745,157.282
C04473=1038.877,41.647,413.378,169.390,38.745,157.282
C04474=1038.871,41.398,413.395,169.388,38.744,157.282
C04475=1038.865,41.148,413.412,169.385,38.744,157.282
C04476=1038.859,40.899,413.428,169.383,38.743,157.281
C04477=1038.852,40.650,413.445,169.381,38.743,157.281
C04478=1038.846,40.400,413.462,169.379,38.742,157.281
C04479=1038.839,40.151,413.479,169.377,38.742,157.281
C04480=1038.833,39.902,413.495,169.375,38.742,157.281
C04481=1038.827,39.653,413.512,169.373,38.741,157.281
C04482=1038.820,39.403,413.529,169.371,38.741,157.281
C04483=1038.814,39.153,413.545,169.370,38.740,157.280
C04484=1038.808,38.905,413.562,169.367,38.740,157.280
C04485=1038.801,38.655,413.579,169.365,38.739,157.280
C04486=1038.795,38.406,413.596,169.363,38.739,157.280
C04487=1038.789,38.157,413.612,169.361,38.739,157.280
C04488=1038.783,37.907,413.628,169.359,38.738,157.280
C04489=1038.776,37.658,413.645,169.357,38.738,157.280
C04490=1038.770,37.408,413.662,169.355,38.737,157.280
C04491=1038.764,37.158,413.678,169.353,38.737,157.279
C04492=1038.758,36.910,413.695,169.351,38.737,157.279
C04493=1038.751,36.660,413.712,169.348,38.736,157.279
C04494=1038.745,36.410,413.728,169.346,38.736,157.279
C04495=1038.738,36.161,413.744,169.344,38.735,157.279
C04496=1038.732,35.912,413.761,169.342,38.735,157.279
C04497=1038.726,35.662,413.777,169.340,38.735,157.279
C04498=1038.720,35.413,413.794,169.339,38.734,157.279
C04499=1038.713,35.163,413.810,169.337,38.734,157.278
C04500=1038.706,34.915,413.827,169.335,38.734,157.278
C04501=1038.700,34.665,413.843,169.333,38.733,157.278
C04502=1038.694,34.415,413.860,169.331,38.733,157.278
C04503=1038.688,34.166,413.876,169.328,38.732,157.278
C04504=1038.681,33.917,413.893,169.326,38.732,157.278
C04505=1038.674,33.667,413.909,169.324,38.732,157.278
C04506=1038.668,33.418,413.925,169.322,38.731,157.278
C04507=1038.662,33.169,413.941,169.320,38.731,157.277
C04508=1038.656,32.919,413.958,169.318,38.731,157.277
C04509=1038.650,32.669,413.974,169.316,38.730,157.277
C04510=1038.643,32.421,413.991,169.314,38.730,157.277
C04511=1038.637,32.172,414.007,169.312,38.729,157.277
C04512=1038.630,31.922,414.023,169.310,38.729,157.277
C04513=1038.624,31.672,414.040,169.308,38.729,157.277
C04514=1038.618,31.423,414.056,169.305,38.728,157.277
C04515=1038.612,31.174,414.072,169.303,38.728,157.276
C04516=1038.605,30.924,414.088,169.301,38.728,157.276
C04517=1038.599,30.675,414.105,169.299,38.727,157.276
C04518=1038.593,30.426,414.121,169.297,38.727,157.276
C04519=1038.586,30.177,414.137,169.295,38.726,157.276
C04520=1038.580,29.927,414.154,169.294,38.726,157.276
C04521=1038.574,29.677,414.170,169.292,38.726,157.276
C04522=1038.568,29.428,414.186,169.290,38.725,157.276
C04523=1038.561,29.179,414.202,169.287,38.725,157.276
C04524=1038.554,28.892,414.222,169.284,38.724,157.275
C04525=1038.547,28.605,414.239,169.282,38.724,157.275
C04526=1038.539,28.318,414.258,169.280,38.723,157.275
C04527=1038.532,28.032,414.277,169.278,38.723,157.275
C04528=1038.526,27.783,414.293,169.276,38.723,157.275
C04529=1038.519,27.533,414.310,169.274,38.722,157.275
C04530=1038.513,27.284,414.325,169.272,38.722,157.275
C04531=1038.507,27.034,414.342,169.270,38.722,157.275
C04532=1038.500,26.785,414.357,169.268,38.721,157.274
C04533=1038.494,26.535,414.373,169.265,38.721,157.274
C04534=1038.488,26.285,414.389,169.263,38.721,157.274
C04535=1038.481,26.036,414.405,169.261,38.720,157.274
C04536=1038.475,25.787,414.421,169.259,38.720,157.274
C04537=1038.469,25.538,414.437,169.257,38.720,157.274
C04538=1038.462,25.288,414.454,169.255,38.720,157.274
C04539=1038.455,25.039,414.469,169.253,38.719,157.274
C04540=1038.449,24.790,414.485,169.251,38.719,157.274
C04541=1038.443,24.540,414.502,169.249,38.719,157.273
C04542=1038.437,24.291,414.517,169.247,38.718,157.273
C04543=1038.431,24.041,414.533,169.244,38.718,157.273
C04544=1038.424,23.791,414.549,169.242,38.718,157.273
C04545=1038.418,23.542,414.565,169.240,38.717,157.273
C04546=1038.411,23.293,414.581,169.238,38.717,157.273
C04547=1038.405,23.044,414.597,169.236,38.717,157.273
C04548=1038.399,22.795,414.613,169.234,38.716,157.273
C04549=1038.393,22.545,414.629,169.232,38.716,157.272
C04550=1038.386,22.295,414.644,169.230,38.716,157.272
C04551=1038.380,22.046,414.661,169.228,38.715,157.272
C04552=1038.373,21.797,414.676,169.226,38.715,157.272
C04553=1038.367,21.547,414.693,169.224,38.715,157.272
C04554=1038.360,21.298,414.708,169.222,38.714,157.272
C04555=1038.355,21.048,414.724,169.219,38.714,157.272
C04556=1038.348,20.799,414.739,169.217,38.713,157.272
C04557=1038.342,20.550,414.756,169.215,38.713,157.272
C04558=1038.336,20.300,414.772,169.213,38.713,157.271
C04559=1038.329,20.050,414.787,169.211,38.712,157.271
C04560=1038.323,19.801,414.804,169.209,38.712,157.271
C04561=1038.316,19.552,414.819,169.207,38.712,157.271
C04562=1038.310,19.302,414.834,169.205,38.711,157.271
C04563=1038.304,19.053,414.850,169.203,38.711,157.271
C04564=1038.297,18.804,414.866,169.201,38.711,157.271
C04565=1038.291,18.554,414.881,169.198,38.710,157.271
C04566=1038.285,18.305,414.897,169.196,38.711,157.271
C04567=1038.278,18.056,414.913,169.194,38.710,157.270
C04568=1038.273,17.806,414.928,169.192,38.709,157.270
C04569=1038.265,17.556,414.944,169.190,38.710,157.270
C04570=1038.259,17.307,414.960,169.188,38.709,157.270
C04571=1038.253,17.057,414.976,169.186,38.709,157.270
C04572=1038.246,16.808,414.991,169.184,38.709,157.270
C04573=1038.240,16.559,415.007,169.182,38.708,157.270
C04574=1038.234,16.309,415.023,169.180,38.708,157.270
C04575=1038.227,16.060,415.038,169.178,38.708,157.270
C04576=1038.222,15.810,415.054,169.176,38.707,157.269
C04577=1038.215,15.561,415.069,169.174,38.707,157.269
C04578=1038.208,15.312,415.085,169.171,38.707,157.269
C04579=1038.203,15.062,415.101,169.168,38.706,157.269
C04580=1038.196,14.813,415.116,169.166,38.706,157.269
C04581=1038.190,14.563,415.131,169.164,38.706,157.269
C04582=1038.184,14.314,415.147,169.162,38.705,157.269
C04583=1038.177,14.064,415.162,169.160,38.705,157.269
C04584=1038.171,13.815,415.178,169.158,38.705,157.269
C04585=1038.164,13.565,415.193,169.156,38.705,157.269
C04586=1038.158,13.316,415.209,169.154,38.705,157.268
C04587=1038.152,13.066,415.224,169.152,38.705,157.268
C04588=1038.144,12.781,415.242,169.150,38.704,157.268
C04589=1038.137,12.496,415.260,169.146,38.704,157.268
C04590=1038.130,12.210,415.277,169.144,38.704,157.268
C04591=1038.122,11.925,415.294,169.142,38.703,157.268
C04592=1038.115,11.676,415.310,169.140,38.703,157.268
C04593=1038.109,11.426,415.325,169.137,38.703,157.268
C04594=1038.103,11.177,415.340,169.135,38.703,157.268
C04595=1038.096,10.928,415.355,169.133,38.702,157.268
C04596=1038.090,10.678,415.370,169.131,38.703,157.268
C04597=1038.084,10.429,415.387,169.129,38.702,157.267
C04598=1038.077,10.179,415.402,169.127,38.702,157.267
C04599=1038.071,9.929,415.417,169.125,38.702,157.267
C04600=1038.064,9.680,415.432,169.123,38.702,157.267
C04601=1038.058,9.431,415.447,169.121,38.701,157.267
C04602=1038.051,9.181,415.462,169.118,38.701,157.267
C04603=1038.045,8.932,415.478,169.116,38.701,157.267
C04604=1038.038,8.682,415.493,169.114,38.700,157.267
C04605=1038.032,8.433,415.508,169.112,38.700,157.267
C04606=1038.025,8.183,415.523,169.109,38.700,157.267
C04607=1038.019,7.934,415.538,169.107,38.700,157.266
C04608=1038.013,7.684,415.553,169.105,38.699,157.266
C04609=1038.007,7.434,415.569,169.103,38.700,157.266
C04610=1038.000,7.185,415.584,169.101,38.699,157.266
C04611=1037.994,6.936,415.599,169.099,38.699,157.266
C04612=1037.988,6.687,415.614,169.097,38.699,157.266
C04613=1037.982,6.437,415.629,169.095,38.699,157.266
C04614=1037.975,6.188,415.645,169.093,38.698,157.266
C04615=1037.969,5.938,415.659,169.091,38.698,157.266
C04616=1037.962,5.689,415.674,169.088,38.698,157.266
C04617=1037.956,5.439,415.689,169.086,38.697,157.265
C04618=1037.949,5.190,415.705,169.083,38.697,157.265
C04619=1037.943,4.940,415.720,169.081,38.697,157.265
C04620=1037.936,4.691,415.735,169.079,38.697,157.265
C04621=1037.931,4.442,415.750,169.077,38.696,157.265
C04622=1037.924,4.192,415.764,169.075,38.697,157.265
C04623=1037.917,3.943,415.780,169.073,38.696,157.265
C04624=1037.912,3.693,415.796,169.071,38.696,157.265
C04625=1037.905,3.443,415.811,169.069,38.696,157.265
C04626=1037.899,3.194,415.826,169.067,38.695,157.265
C04627=1037.893,2.944,415.840,169.065,38.695,157.265
C04628=1037.887,2.695,415.855,169.062,38.695,157.264
C04629=1037.881,2.445,415.870,169.059,38.695,157.264
C04630=1037.874,2.196,415.886,169.057,38.694,157.264
C04631=1037.867,1.947,415.901,169.055,38.694,157.264
C04632=1037.861,1.697,415.916,169.053,38.694,157.264
C04633=1037.855,1.447,415.931,169.051,38.694,157.264
C04634=1037.849,1.198,415.945,169.049,38.693,157.264
C04635=1037.843,0.949,415.960,169.047,38.693,157.264
C04636=1037.836,0.699,415.975,169.045,38.693,157.264
C04637=1037.830,0.449,415.990,169.043,38.693,157.264
C04638=1037.824,0.200,416.005,169.041,38.693,157.264
C04639=1037.818,-0.049,416.019,169.038,38.692,157.263
C04640=1037.811,-0.299,416.034,169.036,38.692,157.263
C04641=1037.805,-0.549,416.049,169.033,38.692,157.263
C04642=1037.798,-0.798,416.064,169.031,38.691,157.263
C04643=1037.793,-1.047,416.079,169.029,38.691,157.263
C04644=1037.786,-1.297,416.094,169.027,38.691,157.263
C04645=1037.780,-1.546,416.109,169.025,38.691,157.263
C04646=1037.773,-1.796,416.124,169.023,38.690,157.263
C04647=1037.768,-2.045,416.138,169.021,38.690,157.263
C04648=1037.761,-2.295,416.153,169.019,38.690,157.262
C04649=1037.755,-2.544,416.168,169.016,38.689,157.262
C04650=1037.749,-2.794,416.183,169.014,38.690,157.262
C04651=1037.743,-3.043,416.198,169.012,38.689,157.262
C04652=1037.736,-3.326,416.215,169.010,38.689,157.262
C04653=1037.728,-3.610,416.232,169.007,38.689,157.262
C04654=1037.721,-3.894,416.248,169.004,38.688,157.262
C04655=1037.714,-4.177,416.265,169.001,38.688,157.262
C04656=1037.708,-4.427,416.280,168.999,38.688,157.262
C04657=1037.701,-4.676,416.294,168.997,38.688,157.262
C04658=1037.695,-4.925,416.309,168.995,38.688,157.262
C04659=1037.689,-5.175,416.324,168.993,38.687,157.261
C04660=1037.682,-5.424,416.338,168.991,38.688,157.261
C04661=1037.676,-5.674,416.352,168.988,38.688,157.261
C04662=1037.670,-5.923,416.367,168.986,38.687,157.261
C04663=1037.663,-6.173,416.382,168.984,38.687,157.261
C04664=1037.656,-6.422,416.396,168.982,38.687,157.261
C04665=1037.650,-6.671,416.411,168.980,38.687,157.261
C04666=1037.644,-6.922,416.425,168.978,38.687,157.261
C04667=1037.637,-7.171,416.439,168.975,38.687,157.261
C04668=1037.631,-7.421,416.454,168.973,38.687,157.261
C04669=1037.625,-7.670,416.469,168.971,38.687,157.261
C04670=1037.618,-7.920,416.482,168.968,38.686,157.261
C04671=1037.612,-8.169,416.497,168.966,38.686,157.261
C04672=1037.606,-8.418,416.512,168.964,38.686,157.260
C04673=1037.599,-8.668,416.526,168.961,38.686,157.260
C04674=1037.593,-8.918,416.541,168.959,38.686,157.260
C04675=1037.587,-9.167,416.555,168.957,38.686,157.260
C04676=1037.580,-9.416,416.569,168.955,38.686,157.260
C04677=1037.574,-9.666,416.584,168.953,38.685,157.260
C04678=1037.568,-9.915,416.598,168.950,38.685,157.260
C04679=1037.561,-10.165,416.613,168.948,38.685,157.260
C04680=1037.555,-10.415,416.627,168.946,38.685,157.260
C04681=1037.549,-10.664,416.641,168.944,38.685,157.260
C04682=1037.542,-10.913,416.656,168.942,38.684,157.260
C04683=1037.536,-11.163,416.670,168.940,38.685,157.260
C04684=1037.530,-11.413,416.685,168.937,38.685,157.260
C04685=1037.523,-11.663,416.698,168.935,38.684,157.259
C04686=1037.518,-11.911,416.713,168.933,38.684,157.259
C04687=1037.511,-12.161,416.728,168.930,38.684,157.259
C04688=1037.505,-12.410,416.741,168.928,38.684,157.259
C04689=1037.499,-12.660,416.756,168.925,38.684,157.259
C04690=1037.492,-12.910,416.770,168.923,38.684,157.259
C04691=1037.486,-13.159,416.784,168.921,38.684,157.259
C04692=1037.480,-13.409,416.799,168.919,38.683,157.259
C04693=1037.473,-13.658,416.812,168.917,38.683,157.259
C04694=1037.467,-13.908,416.827,168.914,38.683,157.259
C04695=1037.461,-14.158,416.842,168.912,38.683,157.259
C04696=1037.454,-14.406,416.856,168.910,38.683,157.259
C04697=1037.448,-14.657,416.870,168.908,38.682,157.258
C04698=1037.442,-14.906,416.884,168.906,38.683,157.258
C04699=1037.436,-15.156,416.898,168.903,38.683,157.258
C04700=1037.430,-15.405,416.913,168.901,38.682,157.258
C04701=1037.423,-15.655,416.926,168.899,38.682,157.258
C04702=1037.417,-15.904,416.941,168.897,38.682,157.258
C04703=1037.410,-16.154,416.954,168.894,38.682,157.258
C04704=1037.403,-16.403,416.969,168.891,38.682,157.258
C04705=1037.398,-16.652,416.983,168.889,38.682,157.258
C04706=1037.391,-16.902,416.996,168.887,38.682,157.258
C04707=1037.385,-17.151,417.011,168.885,38.682,157.258
C04708=1037.378,-17.401,417.024,168.882,38.682,157.258
C04709=1037.372,-17.650,417.038,168.880,38.682,157.258
C04710=1037.366,-17.900,417.053,168.878,38.682,157.258
C04711=1037.360,-18.150,417.066,168.876,38.682,157.257
C04712=1037.353,-18.399,417.080,168.873,38.682,157.257
C04713=1037.347,-18.648,417.094,168.871,38.682,157.257
C04714=1037.340,-18.898,417.108,168.869,38.682,157.257
C04715=1037.334,-19.148,417.123,168.867,38.681,157.257
C04716=1037.327,-19.430,417.138,168.864,38.682,157.257
C04717=1037.320,-19.712,417.154,168.862,38.682,157.257
C04718=1037.313,-19.993,417.169,168.859,38.681,157.257
C04719=1037.306,-20.275,417.185,168.856,38.681,157.257
C04720=1037.299,-20.525,417.199,168.854,38.682,157.257
C04721=1037.292,-20.774,417.213,168.852,38.682,157.257
C04722=1037.286,-21.024,417.227,168.850,38.681,157.257
C04723=1037.280,-21.273,417.240,168.847,38.681,157.257
C04724=1037.274,-21.523,417.254,168.845,38.681,157.257
C04725=1037.267,-21.772,417.268,168.843,38.682,157.257
C04726=1037.261,-22.021,417.282,168.840,38.681,157.256
C04727=1037.255,-22.272,417.296,168.837,38.681,157.256
C04728=1037.249,-22.521,417.309,168.835,38.681,157.256
C04729=1037.242,-22.770,417.323,168.833,38.681,157.256
C04730=1037.236,-23.020,417.337,168.831,38.681,157.256
C04731=1037.229,-23.270,417.351,168.828,38.681,157.256
C04732=1037.223,-23.519,417.364,168.826,38.681,157.256
C04733=1037.218,-23.769,417.378,168.824,38.681,157.256
C04734=1037.211,-24.018,417.392,168.821,38.681,157.256
C04735=1037.204,-24.267,417.406,168.819,38.681,157.256
C04736=1037.198,-24.518,417.420,168.817,38.681,157.256
C04737=1037.192,-24.767,417.433,168.815,38.680,157.256
C04738=1037.186,-25.016,417.447,168.812,38.681,157.256
C04739=1037.180,-25.266,417.461,168.810,38.681,157.256
C04740=1037.174,-25.516,417.474,168.808,38.681,157.256
C04741=1037.167,-25.764,417.488,168.806,38.680,157.256
C04742=1037.161,-26.015,417.502,168.803,38.680,157.255
C04743=1037.155,-26.264,417.516,168.801,38.681,157.255
C04744=1037.148,-26.514,417.529,168.799,38.680,157.255
C04745=1037.143,-26.763,417.543,168.796,38.680,157.255
C04746=1037.136,-27.013,417.556,168.794,38.680,157.255
C04747=1037.129,-27.263,417.570,168.792,38.680,157.255
C04748=1037.123,-27.512,417.583,168.790,38.681,157.255
C04749=1037.116,-27.762,417.597,168.786,38.681,157.255
C04750=1037.111,-28.011,417.611,168.784,38.680,157.255
C04751=1037.105,-28.261,417.624,168.782,38.680,157.255
C04752=1037.098,-28.511,417.638,168.779,38.680,157.255
C04753=1037.092,-28.760,417.651,168.777,38.681,157.255
C04754=1037.086,-29.009,417.664,168.775,38.681,157.255
C04755=1037.079,-29.259,417.678,168.772,38.681,157.255
C04756=1037.072,-29.508,417.691,168.770,38.681,157.255
C04757=1037.066,-29.758,417.704,168.768,38.681,157.255
C04758=1037.059,-30.008,417.718,168.765,38.681,157.255
C04759=1037.053,-30.257,417.731,168.763,38.681,157.255
C04760=1037.047,-30.506,417.744,168.761,38.681,157.255
C04761=1037.040,-30.756,417.758,168.758,38.681,157.254
C04762=1037.034,-31.006,417.771,168.756,38.681,157.254
C04763=1037.028,-31.255,417.784,168.754,38.681,157.254
C04764=1037.022,-31.506,417.798,168.751,38.681,157.254
C04765=1037.016,-31.755,417.811,168.749,38.682,157.254
C04766=1037.010,-32.004,417.825,168.747,38.682,157.254
C04767=1037.003,-32.253,417.838,168.744,38.682,157.254
C04768=1036.997,-32.503,417.852,168.742,38.681,157.254
C04769=1036.990,-32.753,417.865,168.740,38.681,157.254
C04770=1036.984,-33.003,417.877,168.737,38.682,157.254
C04771=1036.978,-33.252,417.891,168.735,38.682,157.254
C04772=1036.971,-33.502,417.904,168.733,38.682,157.254
C04773=1036.965,-33.751,417.918,168.730,38.682,157.254
C04774=1036.959,-34.000,417.931,168.728,38.682,157.254
C04775=1036.952,-34.251,417.944,168.726,38.682,157.254
C04776=1036.946,-34.500,417.957,168.723,38.682,157.254
C04777=1036.940,-34.749,417.970,168.721,38.682,157.254
C04778=1036.934,-34.999,417.984,168.719,38.682,157.254
C04779=1036.928,-35.248,417.997,168.716,38.682,157.254
C04780=1036.921,-35.530,418.012,168.714,38.682,157.254
C04781=1036.914,-35.811,418.026,168.710,38.682,157.254
C04782=1036.906,-36.092,418.041,168.707,38.683,157.254
C04783=1036.900,-36.373,418.056,168.705,38.683,157.253
C04784=1036.893,-36.623,418.070,168.702,38.683,157.253
C04785=1036.887,-36.872,418.083,168.700,38.683,157.253
C04786=1036.881,-37.122,418.096,168.697,38.682,157.253
C04787=1036.875,-37.371,418.109,168.695,38.683,157.253
C04788=1036.869,-37.621,418.122,168.693,38.683,157.253
C04789=1036.863,-37.870,418.135,168.690,38.683,157.253
C04790=1036.856,-38.120,418.148,168.688,38.683,157.253
C04791=1036.850,-38.370,418.162,168.686,38.683,157.253
C04792=1036.844,-38.620,418.174,168.683,38.683,157.253
C04793=1036.838,-38.869,418.187,168.681,38.683,157.253
C04794=1036.831,-39.118,418.201,168.679,38.683,157.253
C04795=1036.825,-39.368,418.213,168.676,38.684,157.253
C04796=1036.818,-39.618,418.226,168.674,38.684,157.253
C04797=1036.812,-39.867,418.239,168.671,38.684,157.253
C04798=1036.806,-40.117,418.252,168.669,38.684,157.253
C04799=1036.800,-40.367,418.265,168.667,38.684,157.253
C04800=1036.793,-40.616,418.277,168.664,38.684,157.253
C04801=1036.787,-40.865,418.290,168.662,38.684,157.253
C04802=1036.780,-41.115,418.304,168.659,38.685,157.253
C04803=1036.774,-41.365,418.316,168.657,38.685,157.253
C04804=1036.767,-41.614,418.329,168.654,38.685,157.253
C04805=1036.761,-41.864,418.341,168.652,38.685,157.253
C04806=1036.755,-42.113,418.355,168.650,38.685,157.253
C04807=1036.749,-42.363,418.367,168.647,38.685,157.253
C04808=1036.743,-42.613,418.380,168.645,38.685,157.253
C04809=1036.736,-42.862,418.392,168.642,38.686,157.252
C04810=1036.730,-43.111,418.406,168.640,38.686,157.253
C04811=1036.724,-43.362,418.419,168.638,38.686,157.253
C04812=1036.717,-43.611,418.432,168.635,38.687,157.252
C04813=1036.711,-43.861,418.444,168.633,38.687,157.252
C04814=1036.705,-44.110,418.457,168.630,38.687,157.252
C04815=1036.699,-44.360,418.470,168.628,38.687,157.252
C04816=1036.693,-44.610,418.482,168.625,38.687,157.252
C04817=1036.686,-44.859,418.495,168.623,38.687,157.252
C04818=1036.680,-45.109,418.507,168.621,38.687,157.252
C04819=1036.674,-45.358,418.521,168.618,38.688,157.252
C04820=1036.667,-45.607,418.533,168.616,38.688,157.252
C04821=1036.661,-45.857,418.545,168.613,38.688,157.252
C04822=1036.655,-46.107,418.558,168.611,38.688,157.252
C04823=1036.649,-46.357,418.571,168.608,38.688,157.252
C04824=1036.642,-46.606,418.583,168.606,38.688,157.252
C04825=1036.636,-46.855,418.596,168.604,38.688,157.252
C04826=1036.630,-47.105,418.609,168.601,38.689,157.252
C04827=1036.624,-47.355,418.621,168.599,38.689,157.252
C04828=1036.617,-47.604,418.634,168.596,38.689,157.252
C04829=1036.611,-47.854,418.647,168.594,38.690,157.252
C04830=1036.606,-48.104,418.659,168.591,38.690,157.252
C04831=1036.599,-48.353,418.672,168.589,38.690,157.252
C04832=1036.593,-48.603,418.684,168.587,38.690,157.252
C04833=1036.587,-48.853,418.697,168.584,38.690,157.252
C04834=1036.581,-49.102,418.709,168.582,38.690,157.252
C04835=1036.574,-49.351,418.722,168.579,38.690,157.252
C04836=1036.568,-49.601,418.735,168.577,38.691,157.252
C04837=1036.562,-49.851,418.747,168.574,38.691,157.252
C04838=1036.555,-50.101,418.759,168.572,38.691,157.252
C04839=1036.549,-50.350,418.772,168.569,38.691,157.252
C04840=1036.543,-50.600,418.785,168.567,38.691,157.252
C04841=1036.537,-50.849,418.797,168.565,38.692,157.252
C04842=1036.531,-51.099,418.810,168.562,38.692,157.252
C04843=1036.524,-51.349,418.821,168.560,38.692,157.252
C04844=1036.517,-51.630,418.836,168.557,38.693,157.252
C04845=1036.510,-51.911,418.849,168.554,38.693,157.252
C04846=1036.503,-52.193,418.862,168.551,38.693,157.252
C04847=1036.495,-52.475,418.877,168.548,38.694,157.252
C04848=1036.489,-52.724,418.889,168.546,38.694,157.252
C04849=1036.483,-52.974,418.901,168.543,38.694,157.252
C04850=1036.476,-53.224,418.913,168.541,38.695,157.252
C04851=1036.469,-53.473,418.925,168.538,38.695,157.252
C04852=1036.463,-53.723,418.938,168.536,38.696,157.252
C04853=1036.457,-53.973,418.950,168.533,38.696,157.252
C04854=1036.450,-54.222,418.962,168.531,38.696,157.252
C04855=1036.445,-54.472,418.974,168.528,38.697,157.252
C04856=1036.438,-54.721,418.986,168.526,38.697,157.252
C04857=1036.432,-54.971,418.998,168.523,38.698,157.252
C04858=1036.426,-55.221,419.010,168.520,38.698,157.252
C04859=1036.419,-55.470,419.022,168.518,38.699,157.252
C04860=1036.412,-55.720,419.034,168.515,38.699,157.252
C04861=1036.406,-55.970,419.047,168.513,38.699,157.252
C04862=1036.400,-56.219,419.059,168.510,38.700,157.252
C04863=1036.393,-56.469,419.071,168.508,38.700,157.252
C04864=1036.387,-56.719,419.083,168.505,38.700,157.252
C04865=1036.381,-56.968,419.095,168.503,38.701,157.252
C04866=1036.375,-57.217,419.107,168.500,38.701,157.252
C04867=1036.369,-57.467,419.119,168.498,38.701,157.252
C04868=1036.362,-57.717,419.131,168.495,38.702,157.252
C04869=1036.356,-57.967,419.143,168.493,38.702,157.252
C04870=1036.350,-58.217,419.155,168.490,38.702,157.252
C04871=1036.344,-58.466,419.167,168.488,38.703,157.252
C04872=1036.337,-58.715,419.179,168.485,38.703,157.252
C04873=1036.331,-58.965,419.191,168.483,38.703,157.252
C04874=1036.324,-59.215,419.203,168.480,38.704,157.252
C04875=1036.318,-59.465,419.214,168.477,38.704,157.252
C04876=1036.312,-59.714,419.226,168.475,38.704,157.252
C04877=1036.306,-59.964,419.239,168.472,38.705,157.252
C04878=1036.300,-60.213,419.251,168.470,38.705,157.252
C04879=1036.293,-60.463,419.263,168.467,38.705,157.252
C04880=1036.287,-60.713,419.275,168.465,38.706,157.252
C04881=1036.281,-60.962,419.286,168.462,38.706,157.252
C04882=1036.275,-61.212,419.298,168.460,38.706,157.252
C04883=1036.268,-61.461,419.310,168.457,38.707,157.252
C04884=1036.262,-61.711,419.322,168.455,38.707,157.252
C04885=1036.256,-61.961,419.334,168.452,38.708,157.252
C04886=1036.250,-62.210,419.345,168.449,38.708,157.252
C04887=1036.244,-62.460,419.358,168.447,38.709,157.252
C04888=1036.237,-62.710,419.370,168.444,38.709,157.252
C04889=1036.231,-62.959,419.381,168.442,38.709,157.252
C04890=1036.225,-63.209,419.393,168.439,38.710,157.252
C04891=1036.219,-63.459,419.405,168.437,38.710,157.252
C04892=1036.212,-63.709,419.416,168.435,38.711,157.252
C04893=1036.206,-63.958,419.428,168.433,38.711,157.252
C04894=1036.200,-64.207,419.440,168.430,38.712,157.252
C04895=1036.194,-64.457,419.453,168.428,38.712,157.252
C04896=1036.188,-64.707,419.463,168.425,38.712,157.252
C04897=1036.181,-64.956,419.475,168.422,38.713,157.252
C04898=1036.176,-65.206,419.488,168.420,38.713,157.252
C04899=1036.170,-65.455,419.499,168.417,38.713,157.252
C04900=1036.163,-65.705,419.511,168.415,38.714,157.252
C04901=1036.157,-65.955,419.522,168.412,38.714,157.252
C04902=1036.152,-66.204,419.534,168.410,38.714,157.252
C04903=1036.145,-66.454,419.546,168.407,38.715,157.252
C04904=1036.139,-66.704,419.557,168.405,38.715,157.252
C04905=1036.133,-66.953,419.569,168.402,38.716,157.252
C04906=1036.126,-67.203,419.580,168.399,38.716,157.252
C04907=1036.120,-67.453,419.593,168.397,38.716,157.252
C04908=1036.113,-67.748,419.606,168.394,38.717,157.252
C04909=1036.106,-68.044,419.620,168.391,38.717,157.252
C04910=1036.098,-68.339,419.634,168.388,38.718,157.252
C04911=1036.091,-68.634,419.647,168.385,38.718,157.252
C04912=1036.086,-68.885,419.659,168.382,38.718,157.252
C04913=1036.079,-69.134,419.671,168.380,38.719,157.252
C04914=1036.073,-69.384,419.682,168.377,38.719,157.252
C04915=1036.067,-69.633,419.694,168.374,38.720,157.252
C04916=1036.061,-69.883,419.705,168.372,38.720,157.252
C04917=1036.055,-70.133,419.718,168.369,38.720,157.252
C04918=1036.049,-70.382,419.728,168.367,38.721,157.252
C04919=1036.043,-70.632,419.740,168.364,38.721,157.252
C04920=1036.036,-70.882,419.752,168.362,38.722,157.252
C04921=1036.030,-71.131,419.763,168.359,38.722,157.252
C04922=1036.025,-71.381,419.775,168.356,38.722,157.252
C04923=1036.019,-71.631,419.786,168.354,38.723,157.252
C04924=1036.013,-71.874,419.798,168.351,38.723,157.252
C04925=1036.006,-72.117,419.809,168.349,38.723,157.252
C04926=1036.000,-72.361,419.820,168.346,38.724,157.252
C04927=1035.995,-72.603,419.831,168.344,38.724,157.252
C04928=1035.990,-72.847,419.842,168.341,38.725,157.252
C04929=1035.984,-73.091,419.853,168.339,38.725,157.252
C04930=1035.978,-73.334,419.864,168.336,38.725,157.252
C04931=1035.972,-73.577,419.875,168.334,38.726,157.252
C04932=1035.965,-73.827,419.887,168.331,38.726,157.252
C04933=1035.959,-74.077,419.898,168.328,38.727,157.252
C04934=1035.953,-74.326,419.909,168.326,38.727,157.252
C04935=1035.947,-74.576,419.921,168.324,38.728,157.252
C04936=1035.941,-74.825,419.932,168.322,38.728,157.252
C04937=1035.935,-75.076,419.943,168.319,38.729,157.252
C04938=1035.929,-75.325,419.954,168.316,38.730,157.252
C04939=1035.922,-75.575,419.966,168.314,38.730,157.252
C04940=1035.917,-75.824,419.977,168.311,38.731,157.252
C04941=1035.910,-76.074,419.988,168.308,38.731,157.252
C04942=1035.904,-76.324,419.999,168.306,38.732,157.252
C04943=1035.898,-76.574,420.010,168.303,38.733,157.252
C04944=1035.892,-76.823,420.022,168.300,38.733,157.252
C04945=1035.886,-77.072,420.033,168.298,38.734,157.252
C04946=1035.879,-77.322,420.044,168.295,38.734,157.252
C04947=1035.874,-77.572,420.054,168.293,38.735,157.252
C04948=1035.867,-77.822,420.066,168.290,38.735,157.253
C04949=1035.861,-78.071,420.077,168.287,38.736,157.252
C04950=1035.855,-78.321,420.088,168.285,38.736,157.253
C04951=1035.849,-78.570,420.099,168.282,38.737,157.253
C04952=1035.843,-78.821,420.111,168.279,38.737,157.253
C04953=1035.837,-79.070,420.121,168.277,38.738,157.253
C04954=1035.831,-79.320,420.132,168.274,38.738,157.253
C04955=1035.825,-79.570,420.144,168.271,38.739,157.253
C04956=1035.818,-79.819,420.154,168.270,38.740,157.253
C04957=1035.812,-80.069,420.165,168.267,38.740,157.253
C04958=1035.806,-80.319,420.176,168.264,38.741,157.253
C04959=1035.800,-80.569,420.187,168.262,38.742,157.253
C04960=1035.794,-80.818,420.198,168.259,38.743,157.253
C04961=1035.788,-81.068,420.208,168.256,38.743,157.253
C04962=1035.781,-81.318,420.220,168.254,38.744,157.253
C04963=1035.775,-81.567,420.230,168.251,38.744,157.253
C04964=1035.769,-81.817,420.241,168.248,38.745,157.253
C04965=1035.763,-82.067,420.252,168.246,38.746,157.253
C04966=1035.756,-82.316,420.262,168.243,38.746,157.253
C04967=1035.750,-82.566,420.274,168.240,38.747,157.253
C04968=1035.744,-82.815,420.284,168.237,38.748,157.253
C04969=1035.737,-83.065,420.295,168.235,38.749,157.253
C04970=1035.731,-83.315,420.306,168.232,38.749,157.253
C04971=1035.725,-83.564,420.316,168.229,38.750,157.253
C04972=1035.718,-83.849,420.329,168.227,38.750,157.254
C04973=1035.711,-84.134,420.341,168.224,38.751,157.254
C04974=1035.704,-84.419,420.353,168.221,38.752,157.254
C04975=1035.697,-84.703,420.365,168.218,38.753,157.254
C04976=1035.691,-84.954,420.376,168.215,38.754,157.254
C04977=1035.685,-85.204,420.387,168.213,38.755,157.254
C04978=1035.678,-85.453,420.397,168.210,38.755,157.254
C04979=1035.672,-85.703,420.408,168.207,38.756,157.254
C04980=1035.666,-85.953,420.419,168.204,38.756,157.254
C04981=1035.660,-86.202,420.430,168.202,38.757,157.254
C04982=1035.654,-86.453,420.440,168.199,38.758,157.254
C04983=1035.647,-86.702,420.450,168.196,38.759,157.254
C04984=1035.642,-86.951,420.461,168.194,38.760,157.254
C04985=1035.636,-87.201,420.472,168.191,38.760,157.254
C04986=1035.629,-87.451,420.483,168.189,38.761,157.254
C04987=1035.623,-87.701,420.493,168.186,38.762,157.254
C04988=1035.618,-87.950,420.504,168.184,38.762,157.254
C04989=1035.610,-88.200,420.514,168.181,38.763,157.255
C04990=1035.605,-88.450,420.525,168.178,38.764,157.255
C04991=1035.599,-88.699,420.535,168.176,38.765,157.255
C04992=1035.593,-88.949,420.546,168.173,38.765,157.255
C04993=1035.587,-89.198,420.557,168.170,38.766,157.255
C04994=1035.580,-89.448,420.567,168.167,38.767,157.255
C04995=1035.575,-89.698,420.577,168.165,38.767,157.255
C04996=1035.568,-89.947,420.588,168.162,38.768,157.255
C04997=1035.562,-90.197,420.599,168.159,38.769,157.255
C04998=1035.556,-90.447,420.609,168.158,38.770,157.255
C04999=1035.550,-90.697,420.619,168.154,38.770,157.255
C05000=1035.544,-90.946,420.630,168.152,38.771,157.255
C05001=1035.538,-91.196,420.640,168.149,38.772,157.255
C05002=1035.532,-91.446,420.651,168.147,38.772,157.255
C05003=1035.525,-91.696,420.661,168.144,38.773,157.255
C05004=1035.520,-91.946,420.672,168.141,38.774,157.255
C05005=1035.514,-92.195,420.682,168.139,38.775,157.256
C05006=1035.507,-92.444,420.693,168.136,38.775,157.255
C05007=1035.502,-92.694,420.703,168.133,38.776,157.256
C05008=1035.496,-92.944,420.713,168.130,38.777,157.256
C05009=1035.490,-93.194,420.723,168.128,38.778,157.256
C05010=1035.483,-93.444,420.734,168.125,38.778,157.256
C05011=1035.477,-93.693,420.745,168.122,38.779,157.256
C05012=1035.471,-93.943,420.754,168.120,38.780,157.256
C05013=1035.465,-94.192,420.765,168.118,38.781,157.256
C05014=1035.460,-94.443,420.775,168.115,38.782,157.256
C05015=1035.453,-94.692,420.786,168.112,38.782,157.256
C05016=1035.448,-94.942,420.796,168.110,38.783,157.256
C05017=1035.442,-95.191,420.806,168.107,38.784,157.256
C05018=1035.436,-95.441,420.816,168.104,38.784,157.256
C05019=1035.429,-95.691,420.827,168.101,38.785,157.256
C05020=1035.424,-95.941,420.837,168.099,38.786,157.256
C05021=1035.417,-96.190,420.847,168.096,38.787,157.256
C05022=1035.412,-96.440,420.858,168.093,38.788,157.257
C05023=1035.406,-96.690,420.868,168.090,38.789,157.257
C05024=1035.400,-96.940,420.878,168.088,38.789,157.257
C05025=1035.394,-97.189,420.889,168.085,38.789,157.257
C05026=1035.388,-97.439,420.898,168.083,38.790,157.257
C05027=1035.382,-97.689,420.909,168.080,38.791,157.257
C05028=1035.376,-97.938,420.919,168.078,38.793,157.257
C05029=1035.370,-98.188,420.929,168.075,38.793,157.257
C05030=1035.363,-98.437,420.939,168.072,38.794,157.257
C05031=1035.358,-98.687,420.949,168.069,38.795,157.257
C05032=1035.352,-98.937,420.959,168.067,38.796,157.257
C05033=1035.345,-99.187,420.969,168.064,38.797,157.257
C05034=1035.339,-99.437,420.979,168.061,38.798,157.257
C05035=1035.333,-99.687,420.989,168.058,38.798,157.257
C05036=1035.326,-99.974,421.000,168.056,38.799,157.258
C05037=1035.319,-100.261,421.012,168.053,38.801,157.258
C05038=1035.312,-100.548,421.024,168.050,38.802,157.258
C05039=1035.305,-100.835,421.035,168.046,38.803,157.258
C05040=1035.299,-101.085,421.044,168.044,38.803,157.258
C05041=1035.293,-101.335,421.055,168.041,38.805,157.258
C05042=1035.287,-101.584,421.065,168.038,38.806,157.258
C05043=1035.281,-101.834,421.074,168.035,38.807,157.258
C05044=1035.275,-102.084,421.085,168.032,38.807,157.258
C05045=1035.269,-102.334,421.094,168.031,38.808,157.258
C05046=1035.262,-102.583,421.104,168.028,38.809,157.258
C05047=1035.256,-102.833,421.114,168.025,38.810,157.259
C05048=1035.251,-103.083,421.124,168.022,38.811,157.259
C05049=1035.245,-103.333,421.134,168.020,38.812,157.259
C05050=1035.239,-103.582,421.143,168.017,38.813,157.259
C05051=1035.233,-103.832,421.152,168.014,38.814,157.259
C05052=1035.227,-104.081,421.163,168.011,38.815,157.259
C05053=1035.221,-104.331,421.173,168.008,38.816,157.259
C05054=1035.215,-104.581,421.182,168.006,38.816,157.259
C05055=1035.209,-104.831,421.192,168.004,38.818,157.259
C05056=1035.203,-105.080,421.202,168.001,38.819,157.259
C05057=1035.197,-105.331,421.212,167.998,38.820,157.260
C05058=1035.191,-105.580,421.221,167.995,38.820,157.260
C05059=1035.185,-105.830,421.231,167.993,38.821,157.260
C05060=1035.178,-106.079,421.241,167.990,38.822,157.260
C05061=1035.172,-106.329,421.251,167.987,38.823,157.260
C05062=1035.167,-106.579,421.261,167.984,38.824,157.260
C05063=1035.161,-106.828,421.270,167.981,38.825,157.260
C05064=1035.155,-107.078,421.280,167.980,38.826,157.260
C05065=1035.149,-107.328,421.289,167.977,38.827,157.260
C05066=1035.143,-107.578,421.299,167.974,38.828,157.260
C05067=1035.136,-107.828,421.308,167.971,38.829,157.260
C05068=1035.130,-108.077,421.318,167.968,38.830,157.261
C05069=1035.124,-108.327,421.327,167.965,38.832,157.261
C05070=1035.118,-108.577,421.337,167.963,38.832,157.261
C05071=1035.113,-108.826,421.347,167.960,38.833,157.261
C05072=1035.107,-109.076,421.356,167.958,38.834,157.261
C05073=1035.101,-109.326,421.366,167.955,38.836,157.261
C05074=1035.095,-109.576,421.376,167.952,38.836,157.261
C05075=1035.088,-109.826,421.385,167.949,38.837,157.261
C05076=1035.082,-110.075,421.395,167.947,38.839,157.261
C05077=1035.076,-110.326,421.404,167.944,38.840,157.262
C05078=1035.071,-110.575,421.413,167.941,38.840,157.262
C05079=1035.065,-110.825,421.422,167.938,38.842,157.262
C05080=1035.058,-111.074,421.432,167.936,38.843,157.262
C05081=1035.052,-111.324,421.441,167.933,38.844,157.262
C05082=1035.046,-111.574,421.451,167.931,38.845,157.262
C05083=1035.041,-111.823,421.460,167.928,38.846,157.262
C05084=1035.034,-112.073,421.470,167.925,38.847,157.262
C05085=1035.029,-112.323,421.479,167.922,38.848,157.262
C05086=1035.022,-112.573,421.488,167.919,38.849,157.263
C05087=1035.016,-112.823,421.498,167.916,38.850,157.263
C05088=1035.011,-113.072,421.507,167.915,38.851,157.263
C05089=1035.004,-113.322,421.517,167.912,38.852,157.263
C05090=1034.998,-113.572,421.526,167.909,38.853,157.263
C05091=1034.992,-113.822,421.535,167.906,38.855,157.263
C05092=1034.987,-114.071,421.544,167.903,38.855,157.263
C05093=1034.981,-114.321,421.554,167.900,38.857,157.263
C05094=1034.974,-114.571,421.563,167.898,38.858,157.263
C05095=1034.969,-114.821,421.572,167.895,38.859,157.263
C05096=1034.963,-115.070,421.581,167.893,38.860,157.264
C05097=1034.957,-115.320,421.591,167.890,38.861,157.264
C05098=1034.951,-115.570,421.600,167.887,38.863,157.264
C05099=1034.945,-115.820,421.609,167.884,38.863,157.264
C05100=1034.938,-116.106,421.619,167.881,38.865,157.264
C05101=1034.931,-116.392,421.630,167.878,38.866,157.264
C05102=1034.925,-116.679,421.641,167.874,38.867,157.264
C05103=1034.917,-116.965,421.651,167.872,38.869,157.265
C05104=1034.911,-117.216,421.660,167.869,38.870,157.265
C05105=1034.906,-117.465,421.669,167.866,38.871,157.265
C05106=1034.899,-117.715,421.679,167.864,38.872,157.265
C05107=1034.894,-117.965,421.688,167.861,38.874,157.265
C05108=1034.887,-118.215,421.697,167.858,38.874,157.265
C05109=1034.881,-118.464,421.705,167.856,38.876,157.265
C05110=1034.875,-118.714,421.715,167.853,38.877,157.265
C05111=1034.869,-118.964,421.724,167.850,38.878,157.266
C05112=1034.864,-119.214,421.733,167.847,38.879,157.266
C05113=1034.858,-119.463,421.742,167.844,38.881,157.266
C05114=1034.852,-119.713,421.750,167.842,38.881,157.266
C05115=1034.846,-119.963,421.760,167.839,38.883,157.266
C05116=1034.840,-120.213,421.769,167.836,38.884,157.266
C05117=1034.834,-120.462,421.778,167.834,38.885,157.266
C05118=1034.828,-120.712,421.787,167.831,38.886,157.266
C05119=1034.822,-120.962,421.796,167.828,38.888,157.267
C05120=1034.816,-121.211,421.805,167.825,38.889,157.267
C05121=1034.810,-121.462,421.814,167.822,38.890,157.267
C05122=1034.804,-121.711,421.823,167.820,38.892,157.267
C05123=1034.798,-121.961,421.832,167.818,38.892,157.267
C05124=1034.792,-122.211,421.841,167.815,38.894,157.267
C05125=1034.786,-122.460,421.849,167.812,38.895,157.267
C05126=1034.780,-122.711,421.858,167.809,38.896,157.268
C05127=1034.775,-122.960,421.867,167.806,38.897,157.268
C05128=1034.768,-123.210,421.876,167.803,38.899,157.268
C05129=1034.763,-123.459,421.885,167.800,38.900,157.268
C05130=1034.757,-123.709,421.894,167.798,38.901,157.268
C05131=1034.751,-123.959,421.903,167.796,38.903,157.268
C05132=1034.745,-124.209,421.912,167.793,38.903,157.268
C05133=1034.739,-124.459,421.920,167.790,38.905,157.268
C05134=1034.733,-124.708,421.929,167.787,38.906,157.269
C05135=1034.727,-124.959,421.938,167.784,38.907,157.269
C05136=1034.721,-125.208,421.946,167.782,38.909,157.269
C05137=1034.715,-125.458,421.955,167.779,38.910,157.269
C05138=1034.709,-125.707,421.963,167.776,38.911,157.269
C05139=1034.703,-125.958,421.972,167.773,38.913,157.269
C05140=1034.698,-126.207,421.981,167.770,38.914,157.270
C05141=1034.691,-126.457,421.990,167.768,38.915,157.270
C05142=1034.685,-126.707,421.998,167.766,38.917,157.270
C05143=1034.680,-126.956,422.008,167.763,38.918,157.270
C05144=1034.674,-127.206,422.016,167.760,38.919,157.270
C05145=1034.668,-127.456,422.024,167.757,38.920,157.270
C05146=1034.661,-127.705,422.033,167.754,38.922,157.270
C05147=1034.656,-127.955,422.042,167.751,38.923,157.270
C05148=1034.651,-128.205,422.052,167.749,38.924,157.271
C05149=1034.646,-128.455,422.061,167.746,38.924,157.270
C05150=1034.643,-128.704,422.071,167.744,38.924,157.270
C05151=1034.640,-128.954,422.082,167.742,38.923,157.270
C05152=1034.639,-129.203,422.095,167.740,38.922,157.270
C05153=1034.637,-129.454,422.107,167.738,38.920,157.270
C05154=1034.636,-129.704,422.120,167.735,38.918,157.269
C05155=1034.635,-129.953,422.133,167.734,38.916,157.269
C05156=1034.636,-130.203,422.147,167.731,38.913,157.268
C05157=1034.638,-130.453,422.162,167.730,38.910,157.268
C05158=1034.640,-130.703,422.177,167.728,38.906,157.267
C05159=1034.643,-130.953,422.193,167.727,38.901,157.266
C05160=1034.646,-131.203,422.210,167.726,38.897,157.265
C05161=1034.650,-131.453,422.227,167.725,38.891,157.264
C05162=1034.654,-131.704,422.244,167.723,38.886,157.263
C05163=1034.660,-131.953,422.263,167.722,38.879,157.262
C05164=1034.328,-131.978,421.980,167.673,39.099,157.298
C05165=1034.322,-131.729,421.961,167.674,39.106,157.299
C05166=1034.318,-131.478,421.944,167.675,39.111,157.300
C05167=1034.314,-131.228,421.926,167.677,39.117,157.301
C05168=1034.310,-130.978,421.911,167.678,39.121,157.302
C05169=1034.307,-130.728,421.894,167.680,39.126,157.302
C05170=1034.305,-130.479,421.879,167.681,39.129,157.303
C05171=1034.304,-130.228,421.864,167.683,39.133,157.304
C05172=1034.303,-129.978,421.850,167.685,39.136,157.304
C05173=1034.303,-129.728,421.837,167.687,39.138,157.305
C05174=1034.304,-129.479,421.823,167.689,39.140,157.305
C05175=1034.306,-129.228,421.811,167.691,39.142,157.306
C05176=1034.308,-128.978,421.800,167.693,39.143,157.306
C05177=1034.311,-128.728,421.789,167.695,39.144,157.306
C05178=1034.314,-128.478,421.778,167.698,39.144,157.306
C05179=1034.318,-128.229,421.768,167.700,39.144,157.306
C05180=1034.323,-127.980,421.759,167.703,39.143,157.306
C05181=1034.329,-127.730,421.750,167.706,39.142,157.306
C05182=1034.335,-127.481,421.741,167.709,39.140,157.306
C05183=1034.342,-127.231,421.733,167.712,39.139,157.306
C05184=1034.347,-126.981,421.724,167.714,39.137,157.305
C05185=1034.352,-126.732,421.715,167.716,39.136,157.305
C05186=1034.359,-126.482,421.707,167.719,39.135,157.305
C05187=1034.364,-126.232,421.698,167.722,39.133,157.305
C05188=1034.371,-125.982,421.690,167.725,39.132,157.305
C05189=1034.376,-125.733,421.681,167.728,39.131,157.305
C05190=1034.382,-125.482,421.672,167.731,39.129,157.305
C05191=1034.389,-125.232,421.664,167.733,39.128,157.304
C05192=1034.394,-124.983,421.654,167.736,39.127,157.304
C05193=1034.400,-124.733,421.645,167.739,39.125,157.304
C05194=1034.406,-124.483,421.638,167.742,39.124,157.304
C05195=1034.412,-124.234,421.628,167.745,39.123,157.304
C05196=1034.418,-123.984,421.620,167.748,39.121,157.304
C05197=1034.424,-123.734,421.610,167.749,39.120,157.304
C05198=1034.430,-123.485,421.602,167.752,39.119,157.303
C05199=1034.436,-123.234,421.593,167.755,39.118,157.303
C05200=1034.441,-122.985,421.584,167.758,39.116,157.303
C05201=1034.447,-122.735,421.575,167.761,39.115,157.303
C05202=1034.454,-122.485,421.566,167.764,39.114,157.303
C05203=1034.459,-122.236,421.558,167.766,39.113,157.303
C05204=1034.466,-121.986,421.548,167.769,39.111,157.303
C05205=1034.471,-121.736,421.540,167.772,39.110,157.302
C05206=1034.477,-121.486,421.531,167.775,39.109,157.302
C05207=1034.484,-121.236,421.522,167.777,39.107,157.302
C05208=1034.489,-120.986,421.513,167.780,39.106,157.302
C05209=1034.495,-120.737,421.504,167.782,39.105,157.302
C05210=1034.500,-120.487,421.495,167.785,39.103,157.302
C05211=1034.507,-120.237,421.486,167.788,39.103,157.302
C05212=1034.513,-119.988,421.477,167.791,39.101,157.302
C05213=1034.519,-119.738,421.468,167.794,39.100,157.301
C05214=1034.525,-119.488,421.459,167.797,39.099,157.301
C05215=1034.530,-119.238,421.450,167.800,39.098,157.301
C05216=1034.537,-118.989,421.441,167.802,39.096,157.301
C05217=1034.543,-118.738,421.432,167.804,39.095,157.301
C05218=1034.548,-118.489,421.423,167.807,39.094,157.301
C05219=1034.555,-118.240,421.414,167.810,39.092,157.301
C05220=1034.560,-117.989,421.405,167.813,39.091,157.301
C05221=1034.566,-117.740,421.396,167.816,39.090,157.300
C05222=1034.572,-117.490,421.387,167.818,39.089,157.300
C05223=1034.579,-117.240,421.378,167.821,39.087,157.300
C05224=1034.585,-116.990,421.368,167.824,39.087,157.300
C05225=1034.591,-116.704,421.358,167.827,39.085,157.300
C05226=1034.597,-116.417,421.348,167.830,39.084,157.300
C05227=1034.605,-116.131,421.337,167.834,39.083,157.300
C05228=1034.612,-115.844,421.326,167.836,39.081,157.300
C05229=1034.618,-115.595,421.317,167.839,39.080,157.299
C05230=1034.623,-115.345,421.308,167.842,39.079,157.299
C05231=1034.629,-115.095,421.299,167.845,39.077,157.299
C05232=1034.636,-114.846,421.290,167.847,39.076,157.299
C05233=1034.642,-114.596,421.280,167.850,39.075,157.299
C05234=1034.648,-114.346,421.272,167.853,39.074,157.299
C05235=1034.654,-114.096,421.262,167.855,39.073,157.299
C05236=1034.660,-113.846,421.253,167.858,39.071,157.299
C05237=1034.666,-113.597,421.243,167.861,39.071,157.298
C05238=1034.671,-113.347,421.235,167.864,39.069,157.298
C05239=1034.678,-113.097,421.225,167.866,39.068,157.298
C05240=1034.684,-112.847,421.215,167.869,39.067,157.298
C05241=1034.690,-112.598,421.206,167.872,39.066,157.298
C05242=1034.695,-112.348,421.197,167.875,39.065,157.298
C05243=1034.701,-112.098,421.188,167.877,39.063,157.298
C05244=1034.708,-111.848,421.178,167.880,39.063,157.298
C05245=1034.714,-111.598,421.169,167.883,39.062,157.298
C05246=1034.720,-111.349,421.159,167.885,39.060,157.297
C05247=1034.725,-111.100,421.150,167.888,39.059,157.297
C05248=1034.732,-110.850,421.140,167.891,39.059,157.297
C05249=1034.737,-110.600,421.130,167.894,39.057,157.297
C05250=1034.743,-110.350,421.121,167.896,39.056,157.297
C05251=1034.749,-110.099,421.112,167.899,39.055,157.297
C05252=1034.755,-109.850,421.103,167.902,39.054,157.297
C05253=1034.761,-109.601,421.093,167.904,39.053,157.297
C05254=1034.767,-109.351,421.083,167.907,39.051,157.297
C05255=1034.773,-109.101,421.074,167.910,39.051,157.296
C05256=1034.779,-108.851,421.064,167.913,39.050,157.296
C05257=1034.785,-108.601,421.055,167.915,39.048,157.296
C05258=1034.792,-108.352,421.045,167.918,39.047,157.296
C05259=1034.797,-108.102,421.036,167.921,39.046,157.296
C05260=1034.803,-107.853,421.026,167.923,39.045,157.296
C05261=1034.810,-107.603,421.017,167.926,39.044,157.296
C05262=1034.816,-107.353,421.007,167.929,39.043,157.296
C05263=1034.822,-107.103,420.998,167.932,39.042,157.296
C05264=1034.827,-106.853,420.988,167.935,39.041,157.296
C05265=1034.834,-106.603,420.978,167.938,39.040,157.295
C05266=1034.840,-106.354,420.968,167.939,39.039,157.295
C05267=1034.845,-106.104,420.959,167.942,39.038,157.295
C05268=1034.851,-105.855,420.950,167.945,39.037,157.295
C05269=1034.858,-105.605,420.940,167.948,39.036,157.295
C05270=1034.863,-105.355,420.930,167.951,39.035,157.295
C05271=1034.870,-105.106,420.920,167.954,39.034,157.295
C05272=1034.876,-104.856,420.910,167.956,39.033,157.295
C05273=1034.882,-104.606,420.900,167.959,39.032,157.295
C05274=1034.887,-104.356,420.890,167.961,39.031,157.295
C05275=1034.893,-104.106,420.881,167.964,39.030,157.295
C05276=1034.900,-103.856,420.871,167.967,39.029,157.294
C05277=1034.906,-103.606,420.862,167.969,39.028,157.294
C05278=1034.912,-103.357,420.851,167.972,39.027,157.294
C05279=1034.918,-103.107,420.841,167.975,39.026,157.294
C05280=1034.923,-102.858,420.832,167.978,39.025,157.294
C05281=1034.929,-102.608,420.822,167.981,39.024,157.294
C05282=1034.936,-102.358,420.813,167.982,39.023,157.294
C05283=1034.941,-102.109,420.802,167.985,39.022,157.294
C05284=1034.948,-101.859,420.792,167.988,39.021,157.294
C05285=1034.954,-101.609,420.783,167.991,39.020,157.294
C05286=1034.959,-101.359,420.773,167.994,39.019,157.294
C05287=1034.965,-101.109,420.763,167.997,39.018,157.293
C05288=1034.972,-100.860,420.753,167.999,39.017,157.293
C05289=1034.979,-100.573,420.742,168.003,39.016,157.293
C05290=1034.986,-100.285,420.730,168.006,39.015,157.293
C05291=1034.993,-99.998,420.718,168.008,39.014,157.293
C05292=1035.000,-99.711,420.708,168.011,39.013,157.293
C05293=1035.005,-99.462,420.697,168.014,39.012,157.293
C05294=1035.012,-99.212,420.687,168.017,39.011,157.293
C05295=1035.018,-98.962,420.678,168.020,39.010,157.293
C05296=1035.025,-98.712,420.667,168.022,39.009,157.293
C05297=1035.030,-98.462,420.657,168.025,39.008,157.292
C05298=1035.036,-98.213,420.647,168.028,39.007,157.292
C05299=1035.043,-97.963,420.637,168.031,39.006,157.292
C05300=1035.048,-97.713,420.627,168.034,39.006,157.292
C05301=1035.055,-97.463,420.617,168.035,39.005,157.292
C05302=1035.060,-97.214,420.606,168.038,39.004,157.292
C05303=1035.066,-96.964,420.597,168.041,39.003,157.292
C05304=1035.072,-96.715,420.586,168.044,39.002,157.292
C05305=1035.078,-96.465,420.576,168.046,39.001,157.292
C05306=1035.084,-96.215,420.566,168.049,39.000,157.292
C05307=1035.090,-95.966,420.556,168.052,39.000,157.292
C05308=1035.096,-95.715,420.546,168.055,38.999,157.292
C05309=1035.102,-95.466,420.535,168.058,38.998,157.292
C05310=1035.108,-95.216,420.525,168.060,38.997,157.292
C05311=1035.115,-94.966,420.515,168.063,38.996,157.291
C05312=1035.120,-94.716,420.504,168.065,38.995,157.291
C05313=1035.126,-94.467,420.494,168.068,38.995,157.291
C05314=1035.132,-94.218,420.483,168.070,38.994,157.291
C05315=1035.138,-93.967,420.473,168.073,38.993,157.291
C05316=1035.144,-93.718,420.463,168.076,38.992,157.291
C05317=1035.150,-93.468,420.453,168.079,38.991,157.291
C05318=1035.156,-93.219,420.442,168.081,38.990,157.291
C05319=1035.162,-92.969,420.432,168.084,38.990,157.291
C05320=1035.169,-92.719,420.422,168.087,38.989,157.291
C05321=1035.174,-92.469,420.411,168.089,38.989,157.291
C05322=1035.180,-92.219,420.401,168.092,38.988,157.291
C05323=1035.186,-91.970,420.390,168.095,38.987,157.291
C05324=1035.192,-91.720,420.380,168.097,38.986,157.291
C05325=1035.198,-91.471,420.370,168.099,38.985,157.291
C05326=1035.205,-91.221,420.359,168.102,38.984,157.291
C05327=1035.211,-90.971,420.349,168.105,38.983,157.290
C05328=1035.216,-90.721,420.338,168.108,38.983,157.290
C05329=1035.222,-90.472,420.327,168.110,38.982,157.290
C05330=1035.228,-90.222,420.318,168.113,38.981,157.290
C05331=1035.235,-89.972,420.306,168.116,38.980,157.290
C05332=1035.241,-89.723,420.296,168.119,38.979,157.290
C05333=1035.247,-89.473,420.286,168.121,38.979,157.290
C05334=1035.252,-89.223,420.275,168.124,38.978,157.290
C05335=1035.259,-88.974,420.265,168.127,38.977,157.290
C05336=1035.265,-88.724,420.254,168.129,38.977,157.290
C05337=1035.271,-88.474,420.244,168.131,38.976,157.290
C05338=1035.277,-88.225,420.233,168.134,38.975,157.290
C05339=1035.283,-87.975,420.222,168.137,38.974,157.290
C05340=1035.290,-87.725,420.212,168.140,38.973,157.290
C05341=1035.295,-87.475,420.201,168.142,38.972,157.290
C05342=1035.302,-87.226,420.191,168.145,38.972,157.290
C05343=1035.308,-86.976,420.180,168.148,38.971,157.290
C05344=1035.314,-86.726,420.169,168.150,38.971,157.290
C05345=1035.320,-86.476,420.160,168.153,38.970,157.289
C05346=1035.326,-86.227,420.149,168.156,38.969,157.289
C05347=1035.333,-85.977,420.138,168.159,38.968,157.289
C05348=1035.339,-85.728,420.127,168.160,38.967,157.289
C05349=1035.344,-85.478,420.116,168.163,38.966,157.289
C05350=1035.351,-85.228,420.106,168.166,38.966,157.289
C05351=1035.357,-84.978,420.095,168.169,38.965,157.289
C05352=1035.363,-84.729,420.085,168.171,38.965,157.289
C05353=1035.370,-84.443,420.072,168.174,38.964,157.289
C05354=1035.377,-84.159,420.060,168.178,38.963,157.289
C05355=1035.384,-83.874,420.047,168.181,38.962,157.289
C05356=1035.391,-83.589,420.035,168.184,38.961,157.289
C05357=1035.398,-83.340,420.025,168.186,38.960,157.289
C05358=1035.404,-83.090,420.014,168.189,38.959,157.289
C05359=1035.410,-82.840,420.003,168.192,38.959,157.289
C05360=1035.416,-82.590,419.993,168.195,38.958,157.289
C05361=1035.422,-82.340,419.982,168.196,38.957,157.288
C05362=1035.429,-82.091,419.972,168.199,38.956,157.288
C05363=1035.435,-81.841,419.961,168.202,38.956,157.288
C05364=1035.441,-81.591,419.950,168.205,38.955,157.288
C05365=1035.448,-81.342,419.939,168.207,38.954,157.288
C05366=1035.454,-81.092,419.928,168.210,38.953,157.288
C05367=1035.459,-80.843,419.917,168.213,38.953,157.288
C05368=1035.466,-80.593,419.907,168.215,38.952,157.288
C05369=1035.472,-80.343,419.896,168.218,38.951,157.288
C05370=1035.478,-80.093,419.885,168.221,38.951,157.288
C05371=1035.485,-79.844,419.874,168.224,38.950,157.288
C05372=1035.491,-79.594,419.863,168.226,38.949,157.288
C05373=1035.497,-79.344,419.852,168.229,38.948,157.288
C05374=1035.503,-79.095,419.841,168.232,38.948,157.288
C05375=1035.509,-78.845,419.829,168.233,38.947,157.288
C05376=1035.515,-78.596,419.818,168.236,38.946,157.288
C05377=1035.521,-78.345,419.807,168.239,38.946,157.288
C05378=1035.527,-78.096,419.796,168.241,38.945,157.288
C05379=1035.533,-77.846,419.785,168.244,38.945,157.288
C05380=1035.539,-77.596,419.774,168.247,38.944,157.288
C05381=1035.546,-77.348,419.763,168.249,38.944,157.288
C05382=1035.552,-77.098,419.752,168.252,38.943,157.287
C05383=1035.558,-76.848,419.741,168.254,38.943,157.288
C05384=1035.564,-76.598,419.730,168.257,38.942,157.287
C05385=1035.570,-76.348,419.719,168.260,38.941,157.287
C05386=1035.577,-76.098,419.708,168.262,38.941,157.287
C05387=1035.583,-75.849,419.696,168.265,38.940,157.287
C05388=1035.589,-75.599,419.685,168.268,38.939,157.287
C05389=1035.595,-75.350,419.674,168.270,38.939,157.287
C05390=1035.601,-75.099,419.663,168.273,38.938,157.287
C05391=1035.607,-74.851,419.651,168.276,38.937,157.287
C05392=1035.613,-74.600,419.640,168.278,38.937,157.287
C05393=1035.619,-74.351,419.629,168.281,38.936,157.287
C05394=1035.625,-74.101,419.618,168.283,38.935,157.287
C05395=1035.632,-73.852,419.606,168.285,38.935,157.287
C05396=1035.638,-73.602,419.595,168.288,38.935,157.287
C05397=1035.644,-73.352,419.584,168.291,38.934,157.287
C05398=1035.650,-73.103,419.572,168.293,38.934,157.287
C05399=1035.656,-72.853,419.561,168.296,38.933,157.287
C05400=1035.662,-72.603,419.549,168.298,38.933,157.287
C05401=1035.668,-72.354,419.538,168.301,38.932,157.287
C05402=1035.674,-72.103,419.527,168.304,38.932,157.287
C05403=1035.680,-71.855,419.515,168.306,38.931,157.287
C05404=1035.686,-71.604,419.504,168.309,38.931,157.287
C05405=1035.692,-71.355,419.492,168.311,38.930,157.287
C05406=1035.698,-71.105,419.480,168.314,38.930,157.287
C05407=1035.704,-70.856,419.469,168.317,38.930,157.287
C05408=1035.710,-70.606,419.457,168.319,38.929,157.287
C05409=1035.716,-70.357,419.447,168.322,38.929,157.287
C05410=1035.722,-70.107,419.434,168.324,38.928,157.287
C05411=1035.728,-69.856,419.423,168.327,38.928,157.287
C05412=1035.734,-69.608,419.411,168.330,38.927,157.287
C05413=1035.741,-69.357,419.400,168.332,38.927,157.287
C05414=1035.746,-69.108,419.388,168.335,38.926,157.287
C05415=1035.752,-68.858,419.377,168.337,38.926,157.287
C05416=1035.758,-68.609,419.365,168.340,38.926,157.287
C05417=1035.766,-68.326,419.352,168.343,38.925,157.287
C05418=1035.773,-68.043,419.339,168.346,38.925,157.287
C05419=1035.779,-67.760,419.326,168.349,38.924,157.287
C05420=1035.786,-67.478,419.313,168.352,38.924,157.287
C05421=1035.793,-67.228,419.301,168.354,38.923,157.287
C05422=1035.798,-66.978,419.289,168.357,38.923,157.287
C05423=1035.804,-66.729,419.277,168.359,38.922,157.287
C05424=1035.811,-66.479,419.265,168.362,38.922,157.287
C05425=1035.817,-66.229,419.254,168.365,38.921,157.287
C05426=1035.823,-65.980,419.242,168.367,38.921,157.287
C05427=1035.829,-65.730,419.231,168.370,38.921,157.287
C05428=1035.836,-65.480,419.219,168.371,38.920,157.287
C05429=1035.842,-65.231,419.207,168.374,38.920,157.287
C05430=1035.847,-64.981,419.195,168.376,38.919,157.287
C05431=1035.854,-64.731,419.183,168.379,38.919,157.287
C05432=1035.860,-64.482,419.172,168.382,38.918,157.287
C05433=1035.866,-64.232,419.160,168.384,38.918,157.287
C05434=1035.872,-63.982,419.148,168.387,38.918,157.287
C05435=1035.878,-63.733,419.136,168.389,38.917,157.287
C05436=1035.885,-63.483,419.125,168.392,38.917,157.287
C05437=1035.891,-63.234,419.113,168.394,38.916,157.287
C05438=1035.897,-62.984,419.101,168.397,38.916,157.287
C05439=1035.903,-62.734,419.090,168.400,38.915,157.287
C05440=1035.910,-62.485,419.078,168.402,38.915,157.287
C05441=1035.916,-62.235,419.066,168.405,38.914,157.287
C05442=1035.921,-61.986,419.054,168.407,38.914,157.287
C05443=1035.928,-61.736,419.042,168.410,38.914,157.287
C05444=1035.934,-61.486,419.030,168.412,38.913,157.287
C05445=1035.940,-61.236,419.018,168.415,38.913,157.287
C05446=1035.946,-60.987,419.006,168.418,38.912,157.287
C05447=1035.953,-60.737,418.995,168.420,38.912,157.287
C05448=1035.959,-60.488,418.983,168.423,38.911,157.287
C05449=1035.965,-60.238,418.970,168.425,38.911,157.287
C05450=1035.972,-59.988,418.958,168.428,38.910,157.287
C05451=1035.978,-59.739,418.947,168.430,38.910,157.287
C05452=1035.984,-59.489,418.934,168.433,38.909,157.287
C05453=1035.990,-59.239,418.923,168.435,38.909,157.287
C05454=1035.997,-58.990,418.911,168.438,38.908,157.287
